LIN {X 0,Y 311.811,Z 387.645,A -85,B 0,C 180,E1 -15794.035,E2 -15794.035} C_VEL
LIN {X 0,Y 308.986,Z 387.993,A -85,B 0,C 180,E1 -15795.788,E2 -15795.788} C_VEL
LIN {X 0,Y 306.588,Z 388.29,A -85,B 0,C 180,E1 -15797.209,E2 -15797.209} C_VEL
LIN {X 0,Y 305.556,Z 388.419,A -85,B 0,C 180,E1 -15798.309,E2 -15798.309} C_VEL
LIN {X 0,Y 305.47,Z 388.429,A -85,B 0,C 180,E1 -15798.682,E2 -15798.682} C_VEL
LIN {X 0,Y 305.516,Z 388.429,A -85,B 0,C 180,E1 -15801.603,E2 -15801.603} C_VEL
LIN {X 0,Y 305.458,Z 388.434,A -85,B 0,C 180,E1 -15804.886,E2 -15804.886} C_VEL
LIN {X 0,Y 305.448,Z 388.435,A -85,B 0,C 180,E1 -15808.354,E2 -15808.354} C_VEL
LIN {X 0,Y 305.515,Z 388.427,A -85,B 0,C 180,E1 -15811.113,E2 -15811.113} C_VEL
LIN {X 0,Y 305.566,Z 388.421,A -85,B 0,C 180,E1 -15814.087,E2 -15814.087} C_VEL
LIN {X 0,Y 305.495,Z 388.428,A -85,B 0,C 180,E1 -15818.402,E2 -15818.402} C_VEL
LIN {X 0,Y 305.584,Z 388.421,A -85,B 0,C 180,E1 -15821.217,E2 -15821.217} C_VEL
LIN {X 0,Y 305.643,Z 388.415,A -85,B 0,C 180,E1 -15825.349,E2 -15825.349} C_VEL
LIN {X 0,Y 305.634,Z 388.411,A -85,B 0,C 180,E1 -15829.399,E2 -15829.399} C_VEL
LIN {X 0,Y 305.806,Z 388.39,A -85,B 0,C 180,E1 -15832.074,E2 -15832.074} C_VEL
LIN {X 0,Y 305.684,Z 388.405,A -85,B 0,C 180,E1 -15834.723,E2 -15834.723} C_VEL
LIN {X 0,Y 305.952,Z 388.373,A -85,B 0,C 180,E1 -15838.684,E2 -15838.684} C_VEL
LIN {X 0,Y 305.952,Z 388.369,A -85,B 0,C 180,E1 -15841.316,E2 -15841.316} C_VEL
LIN {X 0,Y 305.846,Z 388.386,A -85,B 0,C 180,E1 -15846.598,E2 -15846.598} C_VEL
LIN {X 0,Y 305.73,Z 388.401,A -85,B 0,C 180,E1 -15849.26,E2 -15849.26} C_VEL
LIN {X 0,Y 305.584,Z 388.416,A -85,B 0,C 180,E1 -15853.296,E2 -15853.296} C_VEL
LIN {X 0,Y 305.587,Z 388.416,A -85,B 0,C 180,E1 -15856.02,E2 -15856.02} C_VEL
LIN {X 0,Y 305.57,Z 388.416,A -85,B 0,C 180,E1 -15859.445,E2 -15859.445} C_VEL
LIN {X 0,Y 305.485,Z 388.432,A -85,B 0,C 180,E1 -15863.042,E2 -15863.042} C_VEL
LIN {X 0,Y 305.548,Z 388.422,A -85,B 0,C 180,E1 -15866.23,E2 -15866.23} C_VEL
LIN {X 0,Y 305.49,Z 388.431,A -85,B 0,C 180,E1 -15869.05,E2 -15869.05} C_VEL
LIN {X 0,Y 305.46,Z 388.429,A -85,B 0,C 180,E1 -15873.517,E2 -15873.517} C_VEL
LIN {X 0,Y 305.493,Z 388.429,A -85,B 0,C 180,E1 -15876.737,E2 -15876.737} C_VEL
LIN {X 0,Y 305.481,Z 388.431,A -85,B 0,C 180,E1 -15880.607,E2 -15880.607} C_VEL
LIN {X 0,Y 305.49,Z 388.427,A -85,B 0,C 180,E1 -15883.644,E2 -15883.644} C_VEL
LIN {X 0,Y 305.481,Z 388.431,A -85,B 0,C 180,E1 -15887.409,E2 -15887.409} C_VEL
LIN {X 0,Y 305.502,Z 388.43,A -85,B 0,C 180,E1 -15891.602,E2 -15891.602} C_VEL
LIN {X 0,Y 305.473,Z 388.437,A -85,B 0,C 180,E1 -15895.466,E2 -15895.466} C_VEL
LIN {X 0,Y 305.506,Z 388.633,A -85,B 0,C 180,E1 -15895.911,E2 -15895.911} C_VEL
LIN {X 0,Y 308.047,Z 399.573,A -85,B 0,C 180,E1 -15899.495,E2 -15899.495} C_VEL
LIN {X 0,Y 310.178,Z 410.065,A -85,B 0,C 180,E1 -15902.748,E2 -15902.748} C_VEL
LIN {X 0,Y 310.534,Z 413.788,A -85,B 0,C 180,E1 -15903.801,E2 -15903.801} C_VEL
LIN {X 0,Y 315.895,Z 444.317,A -85,B 0,C 180,E1 -15905.024,E2 -15905.024} C_VEL
LIN {X 0,Y 317.621,Z 457.948,A -85,B 0,C 180,E1 -15905.499,E2 -15905.499} C_VEL
LIN {X 0,Y 316.051,Z 522.272,A -85,B 0,C 180,E1 -15906.969,E2 -15906.969} C_VEL
LIN {X 0,Y 315.163,Z 535.447,A -85,B 0,C 180,E1 -15907.507,E2 -15907.507} C_VEL
LIN {X 0,Y 314.017,Z 547.561,A -85,B 0,C 180,E1 -15908.243,E2 -15908.243} C_VEL
LIN {X 0,Y 312.578,Z 559.793,A -85,B 0,C 180,E1 -15909.261,E2 -15909.261} C_VEL
LIN {X 0,Y 311.004,Z 571.378,A -85,B 0,C 180,E1 -15910.53,E2 -15910.53} C_VEL
LIN {X 0,Y 309.347,Z 581.811,A -85,B 0,C 180,E1 -15911.969,E2 -15911.969} C_VEL
LIN {X 0,Y 307.998,Z 591.203,A -85,B 0,C 180,E1 -15913.597,E2 -15913.597} C_VEL
LIN {X 0,Y 306.701,Z 599.615,A -85,B 0,C 180,E1 -15915.401,E2 -15915.401} C_VEL
LIN {X 0,Y 305.449,Z 607.058,A -85,B 0,C 180,E1 -15917.374,E2 -15917.374} C_VEL
LIN {X 0,Y 304.634,Z 613.044,A -85,B 0,C 180,E1 -15919.365,E2 -15919.365} C_VEL
LIN {X 0,Y 304.095,Z 617.779,A -85,B 0,C 180,E1 -15921.36,E2 -15921.36} C_VEL
LIN {X 0,Y 303.747,Z 621.398,A -85,B 0,C 180,E1 -15923.357,E2 -15923.357} C_VEL
LIN {X 0,Y 303.638,Z 623.266,A -85,B 0,C 180,E1 -15924.688,E2 -15924.688} C_VEL
LIN {X 0,Y 303.633,Z 624.67,A -85,B 0,C 180,E1 -15926.018,E2 -15926.018} C_VEL
LIN {X 0,Y 303.625,Z 625.672,A -85,B 0,C 180,E1 -15927.347,E2 -15927.347} C_VEL
LIN {X 0,Y 303.623,Z 626.282,A -85,B 0,C 180,E1 -15928.674,E2 -15928.674} C_VEL
LIN {X 0,Y 303.669,Z 626.498,A -85,B 0,C 180,E1 -15930,E2 -15930} C_VEL
LIN {X 0,Y 303.623,Z 626.275,A -85,B 0,C 180,E1 -15931.326,E2 -15931.326} C_VEL
LIN {X 0,Y 303.625,Z 625.661,A -85,B 0,C 180,E1 -15932.653,E2 -15932.653} C_VEL
LIN {X 0,Y 303.631,Z 624.656,A -85,B 0,C 180,E1 -15933.982,E2 -15933.982} C_VEL
LIN {X 0,Y 303.66,Z 622.845,A -85,B 0,C 180,E1 -15935.611,E2 -15935.611} C_VEL
LIN {X 0,Y 303.947,Z 619.055,A -85,B 0,C 180,E1 -15937.974,E2 -15937.974} C_VEL
LIN {X 0,Y 304.399,Z 614.691,A -85,B 0,C 180,E1 -15939.971,E2 -15939.971} C_VEL
LIN {X 0,Y 305.106,Z 609.138,A -85,B 0,C 180,E1 -15941.965,E2 -15941.965} C_VEL
LIN {X 0,Y 306.28,Z 602.219,A -85,B 0,C 180,E1 -15943.941,E2 -15943.941} C_VEL
LIN {X 0,Y 307.676,Z 593.562,A -85,B 0,C 180,E1 -15945.908,E2 -15945.908} C_VEL
LIN {X 0,Y 308.939,Z 584.685,A -85,B 0,C 180,E1 -15947.543,E2 -15947.543} C_VEL
LIN {X 0,Y 310.43,Z 574.952,A -85,B 0,C 180,E1 -15948.992,E2 -15948.992} C_VEL
LIN {X 0,Y 311.972,Z 564.306,A -85,B 0,C 180,E1 -15950.265,E2 -15950.265} C_VEL
LIN {X 0,Y 313.421,Z 552.402,A -85,B 0,C 180,E1 -15951.369,E2 -15951.369} C_VEL
LIN {X 0,Y 314.705,Z 540.018,A -85,B 0,C 180,E1 -15952.225,E2 -15952.225} C_VEL
LIN {X 0,Y 315.735,Z 527.279,A -85,B 0,C 180,E1 -15952.839,E2 -15952.839} C_VEL
LIN {X 0,Y 316.3,Z 513.841,A -85,B 0,C 180,E1 -15953.228,E2 -15953.228} C_VEL
LIN {X 0,Y 317.502,Z 455.967,A -85,B 0,C 180,E1 -15954.535,E2 -15954.535} C_VEL
LIN {X 0,Y 312.848,Z 426.197,A -85,B 0,C 180,E1 -15955.658,E2 -15955.658} C_VEL
LIN {X 0,Y 310.488,Z 413.594,A -85,B 0,C 180,E1 -15956.193,E2 -15956.193} C_VEL
LIN {X 0,Y 309.956,Z 408.943,A -85,B 0,C 180,E1 -15957.568,E2 -15957.568} C_VEL
LIN {X 0,Y 308.048,Z 399.473,A -85,B 0,C 180,E1 -15960.505,E2 -15960.505} C_VEL
LIN {X 0,Y 305.466,Z 388.438,A -85,B 0,C 180,E1 -15964.131,E2 -15964.131} C_VEL
LIN {X 0,Y 305.495,Z 388.432,A -85,B 0,C 180,E1 -15966.736,E2 -15966.736} C_VEL
LIN {X 0,Y 305.455,Z 388.434,A -85,B 0,C 180,E1 -15970.6,E2 -15970.6} C_VEL
LIN {X 0,Y 305.468,Z 388.432,A -85,B 0,C 180,E1 -15973.646,E2 -15973.646} C_VEL
LIN {X 0,Y 305.505,Z 388.429,A -85,B 0,C 180,E1 -15977.403,E2 -15977.403} C_VEL
LIN {X 0,Y 305.506,Z 388.43,A -85,B 0,C 180,E1 -15981.602,E2 -15981.602} C_VEL
LIN {X 0,Y 305.458,Z 388.435,A -85,B 0,C 180,E1 -15984.886,E2 -15984.886} C_VEL
LIN {X 0,Y 305.447,Z 388.434,A -85,B 0,C 180,E1 -15988.354,E2 -15988.354} C_VEL
LIN {X 0,Y 305.516,Z 388.426,A -85,B 0,C 180,E1 -15991.113,E2 -15991.113} C_VEL
LIN {X 0,Y 305.567,Z 388.419,A -85,B 0,C 180,E1 -15994.087,E2 -15994.087} C_VEL
LIN {X 0,Y 305.494,Z 388.427,A -85,B 0,C 180,E1 -15998.402,E2 -15998.402} C_VEL
LIN {X 0,Y 305.584,Z 388.419,A -85,B 0,C 180,E1 -16001.217,E2 -16001.217} C_VEL
LIN {X 0,Y 305.643,Z 388.414,A -85,B 0,C 180,E1 -16005.349,E2 -16005.349} C_VEL
LIN {X 0,Y 305.634,Z 388.408,A -85,B 0,C 180,E1 -16009.4,E2 -16009.4} C_VEL
LIN {X 0,Y 305.806,Z 388.389,A -85,B 0,C 180,E1 -16012.074,E2 -16012.074} C_VEL
LIN {X 0,Y 305.684,Z 388.408,A -85,B 0,C 180,E1 -16014.723,E2 -16014.723} C_VEL
LIN {X 0,Y 305.952,Z 388.37,A -85,B 0,C 180,E1 -16018.684,E2 -16018.684} C_VEL
LIN {X 0,Y 305.952,Z 388.373,A -85,B 0,C 180,E1 -16021.316,E2 -16021.316} C_VEL
LIN {X 0,Y 305.846,Z 388.384,A -85,B 0,C 180,E1 -16026.598,E2 -16026.598} C_VEL
LIN {X 0,Y 305.73,Z 388.4,A -85,B 0,C 180,E1 -16029.26,E2 -16029.26} C_VEL
LIN {X 0,Y 305.584,Z 388.416,A -85,B 0,C 180,E1 -16033.296,E2 -16033.296} C_VEL
LIN {X 0,Y 305.588,Z 388.418,A -85,B 0,C 180,E1 -16036.021,E2 -16036.021} C_VEL
LIN {X 0,Y 305.571,Z 388.414,A -85,B 0,C 180,E1 -16039.445,E2 -16039.445} C_VEL
LIN {X 0,Y 305.485,Z 388.432,A -85,B 0,C 180,E1 -16043.042,E2 -16043.042} C_VEL
LIN {X 0,Y 305.542,Z 388.42,A -85,B 0,C 180,E1 -16046.228,E2 -16046.228} C_VEL
LIN {X 0,Y 305.491,Z 388.431,A -85,B 0,C 180,E1 -16049.05,E2 -16049.05} C_VEL
LIN {X 0,Y 305.46,Z 388.433,A -85,B 0,C 180,E1 -16053.518,E2 -16053.518} C_VEL
LIN {X 0,Y 305.498,Z 388.429,A -85,B 0,C 180,E1 -16056.736,E2 -16056.736} C_VEL
LIN {X 0,Y 305.482,Z 388.431,A -85,B 0,C 180,E1 -16060.607,E2 -16060.607} C_VEL
LIN {X 0,Y 305.49,Z 388.43,A -85,B 0,C 180,E1 -16063.644,E2 -16063.644} C_VEL
LIN {X 0,Y 305.461,Z 388.433,A -85,B 0,C 180,E1 -16067.413,E2 -16067.413} C_VEL
LIN {X 0,Y 305.494,Z 388.43,A -85,B 0,C 180,E1 -16071.601,E2 -16071.601} C_VEL
LIN {X 0,Y 305.462,Z 388.435,A -85,B 0,C 180,E1 -16074.888,E2 -16074.888} C_VEL
LIN {X 0,Y 305.45,Z 388.439,A -85,B 0,C 180,E1 -16078.356,E2 -16078.356} C_VEL
LIN {X 0,Y 305.542,Z 388.49,A -85,B 0,C 180,E1 -16081.68,E2 -16081.68} C_VEL
LIN {X 0,Y 306.681,Z 393.494,A -85,B 0,C 180,E1 -16083.529,E2 -16083.529} C_VEL
LIN {X 0,Y 315.952,Z 416.268,A -85,B 0,C 180,E1 -16084.939,E2 -16084.939} C_VEL
LIN {X 0,Y 317.657,Z 421.102,A -85,B 0,C 180,E1 -16085.203,E2 -16085.203} C_VEL
LIN {X 0,Y 318.311,Z 425.219,A -85,B 0,C 180,E1 -16085.358,E2 -16085.358} C_VEL
LIN {X 0,Y 316.452,Z 500.83,A -85,B 0,C 180,E1 -16087.087,E2 -16087.087} C_VEL
LIN {X 0,Y 315.602,Z 514.574,A -85,B 0,C 180,E1 -16087.67,E2 -16087.67} C_VEL
LIN {X 0,Y 314.661,Z 526.897,A -85,B 0,C 180,E1 -16088.462,E2 -16088.462} C_VEL
LIN {X 0,Y 313.426,Z 538.705,A -85,B 0,C 180,E1 -16089.491,E2 -16089.491} C_VEL
LIN {X 0,Y 311.975,Z 550.046,A -85,B 0,C 180,E1 -16090.765,E2 -16090.765} C_VEL
LIN {X 0,Y 310.648,Z 560.751,A -85,B 0,C 180,E1 -16092.303,E2 -16092.303} C_VEL
LIN {X 0,Y 309.2,Z 569.411,A -85,B 0,C 180,E1 -16093.833,E2 -16093.833} C_VEL
LIN {X 0,Y 307.641,Z 578.311,A -85,B 0,C 180,E1 -16095.784,E2 -16095.784} C_VEL
LIN {X 0,Y 306.435,Z 585.47,A -85,B 0,C 180,E1 -16097.752,E2 -16097.752} C_VEL
LIN {X 0,Y 305.596,Z 590.296,A -85,B 0,C 180,E1 -16099.398,E2 -16099.398} C_VEL
LIN {X 0,Y 304.832,Z 594.983,A -85,B 0,C 180,E1 -16101.381,E2 -16101.381} C_VEL
LIN {X 0,Y 304.35,Z 598.567,A -85,B 0,C 180,E1 -16103.37,E2 -16103.37} C_VEL
LIN {X 0,Y 304.119,Z 600.418,A -85,B 0,C 180,E1 -16104.696,E2 -16104.696} C_VEL
LIN {X 0,Y 303.925,Z 601.811,A -85,B 0,C 180,E1 -16106.022,E2 -16106.022} C_VEL
LIN {X 0,Y 303.682,Z 603.413,A -85,B 0,C 180,E1 -16108.674,E2 -16108.674} C_VEL
LIN {X 0,Y 303.677,Z 603.643,A -85,B 0,C 180,E1 -16110,E2 -16110} C_VEL
LIN {X 0,Y 303.682,Z 603.452,A -85,B 0,C 180,E1 -16111.326,E2 -16111.326} C_VEL
LIN {X 0,Y 303.924,Z 601.901,A -85,B 0,C 180,E1 -16113.978,E2 -16113.978} C_VEL
LIN {X 0,Y 304.118,Z 600.547,A -85,B 0,C 180,E1 -16115.304,E2 -16115.304} C_VEL
LIN {X 0,Y 304.472,Z 598.158,A -85,B 0,C 180,E1 -16116.995,E2 -16116.995} C_VEL
LIN {X 0,Y 305.019,Z 593.81,A -85,B 0,C 180,E1 -16119.281,E2 -16119.281} C_VEL
LIN {X 0,Y 305.887,Z 588.801,A -85,B 0,C 180,E1 -16121.262,E2 -16121.262} C_VEL
LIN {X 0,Y 306.971,Z 582.493,A -85,B 0,C 180,E1 -16123.235,E2 -16123.235} C_VEL
LIN {X 0,Y 308.267,Z 574.597,A -85,B 0,C 180,E1 -16125.199,E2 -16125.199} C_VEL
LIN {X 0,Y 309.691,Z 566.539,A -85,B 0,C 180,E1 -16126.818,E2 -16126.818} C_VEL
LIN {X 0,Y 311.094,Z 556.711,A -85,B 0,C 180,E1 -16128.438,E2 -16128.438} C_VEL
LIN {X 0,Y 312.554,Z 545.645,A -85,B 0,C 180,E1 -16129.882,E2 -16129.882} C_VEL
LIN {X 0,Y 314.119,Z 533.028,A -85,B 0,C 180,E1 -16131.147,E2 -16131.147} C_VEL
LIN {X 0,Y 315.312,Z 520.402,A -85,B 0,C 180,E1 -16132.093,E2 -16132.093} C_VEL
LIN {X 0,Y 316.15,Z 507.737,A -85,B 0,C 180,E1 -16132.764,E2 -16132.764} C_VEL
LIN {X 0,Y 316.692,Z 494.689,A -85,B 0,C 180,E1 -16133.197,E2 -16133.197} C_VEL
LIN {X 0,Y 318.267,Z 423.968,A -85,B 0,C 180,E1 -16134.79,E2 -16134.79} C_VEL
LIN {X 0,Y 316.849,Z 418.647,A -85,B 0,C 180,E1 -16135.041,E2 -16135.041} C_VEL
LIN {X 0,Y 309.15,Z 399.307,A -85,B 0,C 180,E1 -16136.207,E2 -16136.207} C_VEL
LIN {X 0,Y 306.686,Z 393.484,A -85,B 0,C 180,E1 -16136.596,E2 -16136.596} C_VEL
LIN {X 0,Y 305.522,Z 388.43,A -85,B 0,C 180,E1 -16138.51,E2 -16138.51} C_VEL
LIN {X 0,Y 305.443,Z 388.441,A -85,B 0,C 180,E1 -16141.951,E2 -16141.951} C_VEL
LIN {X 0,Y 305.462,Z 388.435,A -85,B 0,C 180,E1 -16145.112,E2 -16145.112} C_VEL
LIN {X 0,Y 305.465,Z 388.434,A -85,B 0,C 180,E1 -16148.532,E2 -16148.532} C_VEL
LIN {X 0,Y 305.461,Z 388.432,A -85,B 0,C 180,E1 -16152.587,E2 -16152.587} C_VEL
LIN {X 0,Y 305.49,Z 388.424,A -85,B 0,C 180,E1 -16156.356,E2 -16156.356} C_VEL
LIN {X 0,Y 305.47,Z 388.429,A -85,B 0,C 180,E1 -16158.682,E2 -16158.682} C_VEL
LIN {X 0,Y 304.799,Z 388.519,A -85,B 0,C 180,E1 -16159.783,E2 -16159.783} C_VEL
LIN {X 0,Y 301.949,Z 388.874,A -85,B 0,C 180,E1 -16161.576,E2 -16161.576} C_VEL
LIN {X 0,Y 299.532,Z 389.174,A -85,B 0,C 180,E1 -16163.03,E2 -16163.03} C_VEL
LIN {X 0,Y 298.489,Z 389.303,A -85,B 0,C 180,E1 -16164.156,E2 -16164.156} C_VEL
LIN {X 0,Y 298.401,Z 389.312,A -85,B 0,C 180,E1 -16164.537,E2 -16164.537} C_VEL
LIN {X 0,Y 298.391,Z 389.314,A -85,B 0,C 180,E1 -16168.791,E2 -16168.791} C_VEL
LIN {X 0,Y 298.458,Z 389.306,A -85,B 0,C 180,E1 -16171.904,E2 -16171.904} C_VEL
LIN {X 0,Y 298.48,Z 389.304,A -85,B 0,C 180,E1 -16174.923,E2 -16174.923} C_VEL
LIN {X 0,Y 298.445,Z 389.311,A -85,B 0,C 180,E1 -16179.315,E2 -16179.315} C_VEL
LIN {X 0,Y 298.532,Z 389.292,A -85,B 0,C 180,E1 -16182.179,E2 -16182.179} C_VEL
LIN {X 0,Y 298.587,Z 389.291,A -85,B 0,C 180,E1 -16184.994,E2 -16184.994} C_VEL
LIN {X 0,Y 298.589,Z 389.287,A -85,B 0,C 180,E1 -16189.146,E2 -16189.146} C_VEL
LIN {X 0,Y 298.752,Z 389.269,A -85,B 0,C 180,E1 -16191.886,E2 -16191.886} C_VEL
LIN {X 0,Y 298.655,Z 389.279,A -85,B 0,C 180,E1 -16194.599,E2 -16194.599} C_VEL
LIN {X 0,Y 298.919,Z 389.249,A -85,B 0,C 180,E1 -16198.653,E2 -16198.653} C_VEL
LIN {X 0,Y 298.919,Z 389.244,A -85,B 0,C 180,E1 -16201.347,E2 -16201.347} C_VEL
LIN {X 0,Y 298.791,Z 389.266,A -85,B 0,C 180,E1 -16206.754,E2 -16206.754} C_VEL
LIN {X 0,Y 298.675,Z 389.278,A -85,B 0,C 180,E1 -16209.481,E2 -16209.481} C_VEL
LIN {X 0,Y 298.547,Z 389.29,A -85,B 0,C 180,E1 -16213.616,E2 -16213.616} C_VEL
LIN {X 0,Y 298.542,Z 389.295,A -85,B 0,C 180,E1 -16216.409,E2 -16216.409} C_VEL
LIN {X 0,Y 298.505,Z 389.295,A -85,B 0,C 180,E1 -16219.655,E2 -16219.655} C_VEL
LIN {X 0,Y 298.452,Z 389.305,A -85,B 0,C 180,E1 -16223.598,E2 -16223.598} C_VEL
LIN {X 0,Y 298.487,Z 389.305,A -85,B 0,C 180,E1 -16226.575,E2 -16226.575} C_VEL
LIN {X 0,Y 298.416,Z 389.31,A -85,B 0,C 180,E1 -16229.642,E2 -16229.642} C_VEL
LIN {X 0,Y 298.391,Z 389.313,A -85,B 0,C 180,E1 -16232.801,E2 -16232.801} C_VEL
LIN {X 0,Y 298.462,Z 389.304,A -85,B 0,C 180,E1 -16236.813,E2 -16236.813} C_VEL
LIN {X 0,Y 298.448,Z 389.306,A -85,B 0,C 180,E1 -16241.251,E2 -16241.251} C_VEL
LIN {X 0,Y 298.414,Z 389.312,A -85,B 0,C 180,E1 -16245.048,E2 -16245.048} C_VEL
LIN {X 0,Y 298.411,Z 389.314,A -85,B 0,C 180,E1 -16248.907,E2 -16248.907} C_VEL
LIN {X 0,Y 298.463,Z 389.309,A -85,B 0,C 180,E1 -16253.188,E2 -16253.188} C_VEL
LIN {X 0,Y 298.446,Z 389.483,A -85,B 0,C 180,E1 -16255.347,E2 -16255.347} C_VEL
LIN {X 0,Y 301.028,Z 400.576,A -85,B 0,C 180,E1 -16259.095,E2 -16259.095} C_VEL
LIN {X 0,Y 303.14,Z 410.847,A -85,B 0,C 180,E1 -16262.376,E2 -16262.376} C_VEL
LIN {X 0,Y 303.577,Z 413.519,A -85,B 0,C 180,E1 -16263.153,E2 -16263.153} C_VEL
LIN {X 0,Y 305.073,Z 419.768,A -85,B 0,C 180,E1 -16263.455,E2 -16263.455} C_VEL
LIN {X 0,Y 309.974,Z 448.85,A -85,B 0,C 180,E1 -16264.633,E2 -16264.633} C_VEL
LIN {X 0,Y 311.143,Z 458.683,A -85,B 0,C 180,E1 -16264.979,E2 -16264.979} C_VEL
LIN {X 0,Y 309.541,Z 522.018,A -85,B 0,C 180,E1 -16266.456,E2 -16266.456} C_VEL
LIN {X 0,Y 308.55,Z 535.952,A -85,B 0,C 180,E1 -16267.042,E2 -16267.042} C_VEL
LIN {X 0,Y 307.29,Z 548.414,A -85,B 0,C 180,E1 -16267.83,E2 -16267.83} C_VEL
LIN {X 0,Y 305.933,Z 559.53,A -85,B 0,C 180,E1 -16268.789,E2 -16268.789} C_VEL
LIN {X 0,Y 304.305,Z 571.114,A -85,B 0,C 180,E1 -16270.084,E2 -16270.084} C_VEL
LIN {X 0,Y 302.586,Z 581.546,A -85,B 0,C 180,E1 -16271.551,E2 -16271.551} C_VEL
LIN {X 0,Y 301.2,Z 590.232,A -85,B 0,C 180,E1 -16273.072,E2 -16273.072} C_VEL
LIN {X 0,Y 300.003,Z 597.968,A -85,B 0,C 180,E1 -16274.72,E2 -16274.72} C_VEL
LIN {X 0,Y 298.722,Z 605.669,A -85,B 0,C 180,E1 -16276.739,E2 -16276.739} C_VEL
LIN {X 0,Y 297.855,Z 610.949,A -85,B 0,C 180,E1 -16278.431,E2 -16278.431} C_VEL
LIN {X 0,Y 297.204,Z 616.073,A -85,B 0,C 180,E1 -16280.472,E2 -16280.472} C_VEL
LIN {X 0,Y 296.786,Z 620.055,A -85,B 0,C 180,E1 -16282.517,E2 -16282.517} C_VEL
LIN {X 0,Y 296.552,Z 622.999,A -85,B 0,C 180,E1 -16284.561,E2 -16284.561} C_VEL
LIN {X 0,Y 296.531,Z 624.403,A -85,B 0,C 180,E1 -16285.923,E2 -16285.923} C_VEL
LIN {X 0,Y 296.55,Z 625.405,A -85,B 0,C 180,E1 -16287.283,E2 -16287.283} C_VEL
LIN {X 0,Y 296.54,Z 626.016,A -85,B 0,C 180,E1 -16288.642,E2 -16288.642} C_VEL
LIN {X 0,Y 296.581,Z 626.232,A -85,B 0,C 180,E1 -16290,E2 -16290} C_VEL
LIN {X 0,Y 296.54,Z 626.008,A -85,B 0,C 180,E1 -16291.358,E2 -16291.358} C_VEL
LIN {X 0,Y 296.55,Z 625.394,A -85,B 0,C 180,E1 -16292.717,E2 -16292.717} C_VEL
LIN {X 0,Y 296.529,Z 624.388,A -85,B 0,C 180,E1 -16294.077,E2 -16294.077} C_VEL
LIN {X 0,Y 296.553,Z 622.872,A -85,B 0,C 180,E1 -16295.523,E2 -16295.523} C_VEL
LIN {X 0,Y 296.888,Z 618.785,A -85,B 0,C 180,E1 -16298.165,E2 -16298.165} C_VEL
LIN {X 0,Y 297.385,Z 614.422,A -85,B 0,C 180,E1 -16300.209,E2 -16300.209} C_VEL
LIN {X 0,Y 298.129,Z 608.868,A -85,B 0,C 180,E1 -16302.249,E2 -16302.249} C_VEL
LIN {X 0,Y 299.376,Z 601.95,A -85,B 0,C 180,E1 -16304.27,E2 -16304.27} C_VEL
LIN {X 0,Y 300.554,Z 594.885,A -85,B 0,C 180,E1 -16305.947,E2 -16305.947} C_VEL
LIN {X 0,Y 301.856,Z 586.37,A -85,B 0,C 180,E1 -16307.618,E2 -16307.618} C_VEL
LIN {X 0,Y 303.328,Z 577.035,A -85,B 0,C 180,E1 -16309.103,E2 -16309.103} C_VEL
LIN {X 0,Y 305.08,Z 565.464,A -85,B 0,C 180,E1 -16310.567,E2 -16310.567} C_VEL
LIN {X 0,Y 306.631,Z 554.068,A -85,B 0,C 180,E1 -16311.69,E2 -16311.69} C_VEL
LIN {X 0,Y 307.927,Z 542.349,A -85,B 0,C 180,E1 -16312.564,E2 -16312.564} C_VEL
LIN {X 0,Y 309.024,Z 529.756,A -85,B 0,C 180,E1 -16313.231,E2 -16313.231} C_VEL
LIN {X 0,Y 309.691,Z 516.923,A -85,B 0,C 180,E1 -16313.665,E2 -16313.665} C_VEL
LIN {X 0,Y 311.047,Z 457.003,A -85,B 0,C 180,E1 -16315.046,E2 -16315.046} C_VEL
LIN {X 0,Y 306.608,Z 428.099,A -85,B 0,C 180,E1 -16316.164,E2 -16316.164} C_VEL
LIN {X 0,Y 303.846,Z 414.488,A -85,B 0,C 180,E1 -16316.768,E2 -16316.768} C_VEL
LIN {X 0,Y 303.518,Z 413.158,A -85,B 0,C 180,E1 -16316.886,E2 -16316.886} C_VEL
LIN {X 0,Y 301.807,Z 403.876,A -85,B 0,C 180,E1 -16319.798,E2 -16319.798} C_VEL
LIN {X 0,Y 299.204,Z 392.71,A -85,B 0,C 180,E1 -16323.503,E2 -16323.503} C_VEL
LIN {X 0,Y 298.424,Z 389.315,A -85,B 0,C 180,E1 -16324.712,E2 -16324.712} C_VEL
LIN {X 0,Y 298.435,Z 389.308,A -85,B 0,C 180,E1 -16327.754,E2 -16327.754} C_VEL
LIN {X 0,Y 298.412,Z 389.314,A -85,B 0,C 180,E1 -16331.256,E2 -16331.256} C_VEL
LIN {X 0,Y 298.414,Z 389.304,A -85,B 0,C 180,E1 -16335.046,E2 -16335.046} C_VEL
LIN {X 0,Y 298.448,Z 389.306,A -85,B 0,C 180,E1 -16338.749,E2 -16338.749} C_VEL
LIN {X 0,Y 298.462,Z 389.306,A -85,B 0,C 180,E1 -16343.187,E2 -16343.187} C_VEL
LIN {X 0,Y 298.391,Z 389.313,A -85,B 0,C 180,E1 -16347.199,E2 -16347.199} C_VEL
LIN {X 0,Y 298.464,Z 389.302,A -85,B 0,C 180,E1 -16351.904,E2 -16351.904} C_VEL
LIN {X 0,Y 298.48,Z 389.304,A -85,B 0,C 180,E1 -16354.924,E2 -16354.924} C_VEL
LIN {X 0,Y 298.444,Z 389.311,A -85,B 0,C 180,E1 -16359.315,E2 -16359.315} C_VEL
LIN {X 0,Y 298.531,Z 389.292,A -85,B 0,C 180,E1 -16362.179,E2 -16362.179} C_VEL
LIN {X 0,Y 298.587,Z 389.29,A -85,B 0,C 180,E1 -16364.994,E2 -16364.994} C_VEL
LIN {X 0,Y 298.589,Z 389.286,A -85,B 0,C 180,E1 -16369.146,E2 -16369.146} C_VEL
LIN {X 0,Y 298.751,Z 389.268,A -85,B 0,C 180,E1 -16371.886,E2 -16371.886} C_VEL
LIN {X 0,Y 298.655,Z 389.283,A -85,B 0,C 180,E1 -16374.599,E2 -16374.599} C_VEL
LIN {X 0,Y 298.919,Z 389.245,A -85,B 0,C 180,E1 -16378.653,E2 -16378.653} C_VEL
LIN {X 0,Y 298.919,Z 389.249,A -85,B 0,C 180,E1 -16381.347,E2 -16381.347} C_VEL
LIN {X 0,Y 298.791,Z 389.264,A -85,B 0,C 180,E1 -16386.754,E2 -16386.754} C_VEL
LIN {X 0,Y 298.675,Z 389.278,A -85,B 0,C 180,E1 -16389.481,E2 -16389.481} C_VEL
LIN {X 0,Y 298.547,Z 389.291,A -85,B 0,C 180,E1 -16393.616,E2 -16393.616} C_VEL
LIN {X 0,Y 298.543,Z 389.298,A -85,B 0,C 180,E1 -16396.409,E2 -16396.409} C_VEL
LIN {X 0,Y 298.506,Z 389.293,A -85,B 0,C 180,E1 -16399.655,E2 -16399.655} C_VEL
LIN {X 0,Y 298.452,Z 389.306,A -85,B 0,C 180,E1 -16403.598,E2 -16403.598} C_VEL
LIN {X 0,Y 298.485,Z 389.301,A -85,B 0,C 180,E1 -16406.575,E2 -16406.575} C_VEL
LIN {X 0,Y 298.416,Z 389.311,A -85,B 0,C 180,E1 -16409.642,E2 -16409.642} C_VEL
LIN {X 0,Y 298.391,Z 389.316,A -85,B 0,C 180,E1 -16412.801,E2 -16412.801} C_VEL
LIN {X 0,Y 298.466,Z 389.304,A -85,B 0,C 180,E1 -16416.814,E2 -16416.814} C_VEL
LIN {X 0,Y 298.449,Z 389.304,A -85,B 0,C 180,E1 -16421.251,E2 -16421.251} C_VEL
LIN {X 0,Y 298.414,Z 389.31,A -85,B 0,C 180,E1 -16425.048,E2 -16425.048} C_VEL
LIN {X 0,Y 298.386,Z 389.316,A -85,B 0,C 180,E1 -16428.913,E2 -16428.913} C_VEL
LIN {X 0,Y 298.464,Z 389.306,A -85,B 0,C 180,E1 -16433.188,E2 -16433.188} C_VEL
LIN {X 0,Y 298.395,Z 389.315,A -85,B 0,C 180,E1 -16437.201,E2 -16437.201} C_VEL
LIN {X 0,Y 298.47,Z 389.31,A -85,B 0,C 180,E1 -16441.138,E2 -16441.138} C_VEL
LIN {X 0,Y 299.603,Z 394.019,A -85,B 0,C 180,E1 -16442.861,E2 -16442.861} C_VEL
LIN {X 0,Y 308.112,Z 414.287,A -85,B 0,C 180,E1 -16444.196,E2 -16444.196} C_VEL
LIN {X 0,Y 311.401,Z 423.085,A -85,B 0,C 180,E1 -16444.712,E2 -16444.712} C_VEL
LIN {X 0,Y 311.875,Z 425.907,A -85,B 0,C 180,E1 -16444.825,E2 -16444.825} C_VEL
LIN {X 0,Y 309.946,Z 501.112,A -85,B 0,C 180,E1 -16446.577,E2 -16446.577} C_VEL
LIN {X 0,Y 309.06,Z 514.851,A -85,B 0,C 180,E1 -16447.17,E2 -16447.17} C_VEL
LIN {X 0,Y 308.092,Z 527.17,A -85,B 0,C 180,E1 -16447.979,E2 -16447.979} C_VEL
LIN {X 0,Y 306.788,Z 538.978,A -85,B 0,C 180,E1 -16449.027,E2 -16449.027} C_VEL
LIN {X 0,Y 305.274,Z 550.318,A -85,B 0,C 180,E1 -16450.325,E2 -16450.325} C_VEL
LIN {X 0,Y 304.06,Z 559.834,A -85,B 0,C 180,E1 -16451.705,E2 -16451.705} C_VEL
LIN {X 0,Y 302.649,Z 567.993,A -85,B 0,C 180,E1 -16453.126,E2 -16453.126} C_VEL
LIN {X 0,Y 301.296,Z 575.848,A -85,B 0,C 180,E1 -16454.787,E2 -16454.787} C_VEL
LIN {X 0,Y 299.886,Z 583.523,A -85,B 0,C 180,E1 -16456.792,E2 -16456.792} C_VEL
LIN {X 0,Y 298.63,Z 590.564,A -85,B 0,C 180,E1 -16459.148,E2 -16459.148} C_VEL
LIN {X 0,Y 297.803,Z 595.252,A -85,B 0,C 180,E1 -16461.176,E2 -16461.176} C_VEL
LIN {X 0,Y 297.301,Z 598.835,A -85,B 0,C 180,E1 -16463.212,E2 -16463.212} C_VEL
LIN {X 0,Y 297.057,Z 600.686,A -85,B 0,C 180,E1 -16464.57,E2 -16464.57} C_VEL
LIN {X 0,Y 296.865,Z 602.078,A -85,B 0,C 180,E1 -16465.927,E2 -16465.927} C_VEL
LIN {X 0,Y 296.598,Z 603.68,A -85,B 0,C 180,E1 -16468.642,E2 -16468.642} C_VEL
LIN {X 0,Y 296.589,Z 603.909,A -85,B 0,C 180,E1 -16470,E2 -16470} C_VEL
LIN {X 0,Y 296.598,Z 603.719,A -85,B 0,C 180,E1 -16471.358,E2 -16471.358} C_VEL
LIN {X 0,Y 296.864,Z 602.167,A -85,B 0,C 180,E1 -16474.073,E2 -16474.073} C_VEL
LIN {X 0,Y 297.057,Z 600.814,A -85,B 0,C 180,E1 -16475.43,E2 -16475.43} C_VEL
LIN {X 0,Y 297.489,Z 597.954,A -85,B 0,C 180,E1 -16477.465,E2 -16477.465} C_VEL
LIN {X 0,Y 298.03,Z 594.076,A -85,B 0,C 180,E1 -16479.501,E2 -16479.501} C_VEL
LIN {X 0,Y 298.94,Z 589.066,A -85,B 0,C 180,E1 -16481.527,E2 -16481.527} C_VEL
LIN {X 0,Y 300.07,Z 582.758,A -85,B 0,C 180,E1 -16483.545,E2 -16483.545} C_VEL
LIN {X 0,Y 301.434,Z 574.861,A -85,B 0,C 180,E1 -16485.552,E2 -16485.552} C_VEL
LIN {X 0,Y 302.903,Z 566.803,A -85,B 0,C 180,E1 -16487.207,E2 -16487.207} C_VEL
LIN {X 0,Y 304.378,Z 556.974,A -85,B 0,C 180,E1 -16488.859,E2 -16488.859} C_VEL
LIN {X 0,Y 305.908,Z 545.907,A -85,B 0,C 180,E1 -16490.333,E2 -16490.333} C_VEL
LIN {X 0,Y 307.524,Z 533.288,A -85,B 0,C 180,E1 -16491.623,E2 -16491.623} C_VEL
LIN {X 0,Y 308.761,Z 520.659,A -85,B 0,C 180,E1 -16492.588,E2 -16492.588} C_VEL
LIN {X 0,Y 309.634,Z 507.991,A -85,B 0,C 180,E1 -16493.271,E2 -16493.271} C_VEL
LIN {X 0,Y 310.199,Z 494.935,A -85,B 0,C 180,E1 -16493.712,E2 -16493.712} C_VEL
LIN {X 0,Y 311.846,Z 425.247,A -85,B 0,C 180,E1 -16495.31,E2 -16495.31} C_VEL
LIN {X 0,Y 310.389,Z 420.239,A -85,B 0,C 180,E1 -16495.565,E2 -16495.565} C_VEL
LIN {X 0,Y 303.195,Z 402.289,A -85,B 0,C 180,E1 -16496.69,E2 -16496.69} C_VEL
LIN {X 0,Y 299.519,Z 393.747,A -85,B 0,C 180,E1 -16497.296,E2 -16497.296} C_VEL
LIN {X 0,Y 298.47,Z 389.308,A -85,B 0,C 180,E1 -16498.991,E2 -16498.991} C_VEL
LIN {X 0,Y 298.395,Z 389.316,A -85,B 0,C 180,E1 -16502.799,E2 -16502.799} C_VEL
LIN {X 0,Y 298.463,Z 389.306,A -85,B 0,C 180,E1 -16506.811,E2 -16506.811} C_VEL
LIN {X 0,Y 298.386,Z 389.315,A -85,B 0,C 180,E1 -16511.087,E2 -16511.087} C_VEL
LIN {X 0,Y 298.414,Z 389.311,A -85,B 0,C 180,E1 -16514.952,E2 -16514.952} C_VEL
LIN {X 0,Y 298.449,Z 389.303,A -85,B 0,C 180,E1 -16518.749,E2 -16518.749} C_VEL
LIN {X 0,Y 298.466,Z 389.303,A -85,B 0,C 180,E1 -16523.186,E2 -16523.186} C_VEL
LIN {X 0,Y 298.401,Z 389.312,A -85,B 0,C 180,E1 -16524.537,E2 -16524.537} C_VEL
LIN {X 0,Y 297.73,Z 389.398,A -85,B 0,C 180,E1 -16525.663,E2 -16525.663} C_VEL
LIN {X 0,Y 294.899,Z 389.749,A -85,B 0,C 180,E1 -16527.498,E2 -16527.498} C_VEL
LIN {X 0,Y 292.498,Z 390.049,A -85,B 0,C 180,E1 -16528.986,E2 -16528.986} C_VEL
LIN {X 0,Y 291.462,Z 390.177,A -85,B 0,C 180,E1 -16530.138,E2 -16530.138} C_VEL
LIN {X 0,Y 291.374,Z 390.186,A -85,B 0,C 180,E1 -16530.528,E2 -16530.528} C_VEL
LIN {X 0,Y 291.411,Z 390.184,A -85,B 0,C 180,E1 -16534.271,E2 -16534.271} C_VEL
LIN {X 0,Y 291.376,Z 390.186,A -85,B 0,C 180,E1 -16537.299,E2 -16537.299} C_VEL
LIN {X 0,Y 291.453,Z 390.178,A -85,B 0,C 180,E1 -16540.27,E2 -16540.27} C_VEL
LIN {X 0,Y 291.535,Z 390.167,A -85,B 0,C 180,E1 -16544.634,E2 -16544.634} C_VEL
LIN {X 0,Y 291.532,Z 390.165,A -85,B 0,C 180,E1 -16548.88,E2 -16548.88} C_VEL
LIN {X 0,Y 291.703,Z 390.149,A -85,B 0,C 180,E1 -16551.688,E2 -16551.688} C_VEL
LIN {X 0,Y 291.625,Z 390.154,A -85,B 0,C 180,E1 -16554.468,E2 -16554.468} C_VEL
LIN {X 0,Y 291.885,Z 390.125,A -85,B 0,C 180,E1 -16558.62,E2 -16558.62} C_VEL
LIN {X 0,Y 291.885,Z 390.12,A -85,B 0,C 180,E1 -16561.38,E2 -16561.38} C_VEL
LIN {X 0,Y 291.74,Z 390.143,A -85,B 0,C 180,E1 -16566.918,E2 -16566.918} C_VEL
LIN {X 0,Y 291.624,Z 390.155,A -85,B 0,C 180,E1 -16569.712,E2 -16569.712} C_VEL
LIN {X 0,Y 291.517,Z 390.165,A -85,B 0,C 180,E1 -16573.951,E2 -16573.951} C_VEL
LIN {X 0,Y 291.481,Z 390.178,A -85,B 0,C 180,E1 -16576.818,E2 -16576.818} C_VEL
LIN {X 0,Y 291.445,Z 390.174,A -85,B 0,C 180,E1 -16579.875,E2 -16579.875} C_VEL
LIN {X 0,Y 291.395,Z 390.185,A -85,B 0,C 180,E1 -16584.206,E2 -16584.206} C_VEL
LIN {X 0,Y 291.421,Z 390.183,A -85,B 0,C 180,E1 -16587.272,E2 -16587.272} C_VEL
LIN {X 0,Y 291.332,Z 390.195,A -85,B 0,C 180,E1 -16590.437,E2 -16590.437} C_VEL
LIN {X 0,Y 291.34,Z 390.188,A -85,B 0,C 180,E1 -16593.699,E2 -16593.699} C_VEL
LIN {X 0,Y 291.395,Z 390.182,A -85,B 0,C 180,E1 -16597.261,E2 -16597.261} C_VEL
LIN {X 0,Y 291.397,Z 390.185,A -85,B 0,C 180,E1 -16600.632,E2 -16600.632} C_VEL
LIN {X 0,Y 291.35,Z 390.192,A -85,B 0,C 180,E1 -16604.39,E2 -16604.39} C_VEL
LIN {X 0,Y 291.35,Z 390.193,A -85,B 0,C 180,E1 -16608.399,E2 -16608.399} C_VEL
LIN {X 0,Y 291.369,Z 390.191,A -85,B 0,C 180,E1 -16611.162,E2 -16611.162} C_VEL
LIN {X 0,Y 291.413,Z 390.28,A -85,B 0,C 180,E1 -16614.742,E2 -16614.742} C_VEL
LIN {X 0,Y 294.139,Z 402.161,A -85,B 0,C 180,E1 -16618.875,E2 -16618.875} C_VEL
LIN {X 0,Y 296.366,Z 413.077,A -85,B 0,C 180,E1 -16622.441,E2 -16622.441} C_VEL
LIN {X 0,Y 298.52,Z 419.743,A -85,B 0,C 180,E1 -16622.831,E2 -16622.831} C_VEL
LIN {X 0,Y 303.615,Z 450.19,A -85,B 0,C 180,E1 -16624.103,E2 -16624.103} C_VEL
LIN {X 0,Y 304.691,Z 459.382,A -85,B 0,C 180,E1 -16624.435,E2 -16624.435} C_VEL
LIN {X 0,Y 303.051,Z 521.765,A -85,B 0,C 180,E1 -16625.921,E2 -16625.921} C_VEL
LIN {X 0,Y 302.034,Z 535.694,A -85,B 0,C 180,E1 -16626.517,E2 -16626.517} C_VEL
LIN {X 0,Y 300.725,Z 548.153,A -85,B 0,C 180,E1 -16627.319,E2 -16627.319} C_VEL
LIN {X 0,Y 299.313,Z 559.267,A -85,B 0,C 180,E1 -16628.296,E2 -16628.296} C_VEL
LIN {X 0,Y 297.615,Z 570.85,A -85,B 0,C 180,E1 -16629.616,E2 -16629.616} C_VEL
LIN {X 0,Y 295.852,Z 581.282,A -85,B 0,C 180,E1 -16631.116,E2 -16631.116} C_VEL
LIN {X 0,Y 294.281,Z 590.63,A -85,B 0,C 180,E1 -16632.8,E2 -16632.8} C_VEL
LIN {X 0,Y 292.875,Z 599.08,A -85,B 0,C 180,E1 -16634.695,E2 -16634.695} C_VEL
LIN {X 0,Y 291.573,Z 606.525,A -85,B 0,C 180,E1 -16636.763,E2 -16636.763} C_VEL
LIN {X 0,Y 290.618,Z 612.51,A -85,B 0,C 180,E1 -16638.845,E2 -16638.845} C_VEL
LIN {X 0,Y 290.005,Z 617.244,A -85,B 0,C 180,E1 -16640.937,E2 -16640.937} C_VEL
LIN {X 0,Y 289.609,Z 620.864,A -85,B 0,C 180,E1 -16643.031,E2 -16643.031} C_VEL
LIN {X 0,Y 289.475,Z 622.828,A -85,B 0,C 180,E1 -16644.513,E2 -16644.513} C_VEL
LIN {X 0,Y 289.475,Z 625.139,A -85,B 0,C 180,E1 -16647.217,E2 -16647.217} C_VEL
LIN {X 0,Y 289.458,Z 625.749,A -85,B 0,C 180,E1 -16648.609,E2 -16648.609} C_VEL
LIN {X 0,Y 289.496,Z 625.965,A -85,B 0,C 180,E1 -16650,E2 -16650} C_VEL
LIN {X 0,Y 289.458,Z 625.742,A -85,B 0,C 180,E1 -16651.391,E2 -16651.391} C_VEL
LIN {X 0,Y 289.475,Z 625.127,A -85,B 0,C 180,E1 -16652.783,E2 -16652.783} C_VEL
LIN {X 0,Y 289.479,Z 622.798,A -85,B 0,C 180,E1 -16655.494,E2 -16655.494} C_VEL
LIN {X 0,Y 289.715,Z 619.752,A -85,B 0,C 180,E1 -16657.667,E2 -16657.667} C_VEL
LIN {X 0,Y 290.158,Z 615.754,A -85,B 0,C 180,E1 -16659.761,E2 -16659.761} C_VEL
LIN {X 0,Y 290.995,Z 609.613,A -85,B 0,C 180,E1 -16662.2,E2 -16662.2} C_VEL
LIN {X 0,Y 292.227,Z 602.918,A -85,B 0,C 180,E1 -16664.271,E2 -16664.271} C_VEL
LIN {X 0,Y 293.71,Z 594.615,A -85,B 0,C 180,E1 -16666.329,E2 -16666.329} C_VEL
LIN {X 0,Y 295.044,Z 586.098,A -85,B 0,C 180,E1 -16668.038,E2 -16668.038} C_VEL
LIN {X 0,Y 296.808,Z 575.587,A -85,B 0,C 180,E1 -16669.719,E2 -16669.719} C_VEL
LIN {X 0,Y 298.659,Z 563.762,A -85,B 0,C 180,E1 -16671.21,E2 -16671.21} C_VEL
LIN {X 0,Y 300.232,Z 551.856,A -85,B 0,C 180,E1 -16672.357,E2 -16672.357} C_VEL
LIN {X 0,Y 301.585,Z 539.467,A -85,B 0,C 180,E1 -16673.247,E2 -16673.247} C_VEL
LIN {X 0,Y 302.711,Z 526.723,A -85,B 0,C 180,E1 -16673.881,E2 -16673.881} C_VEL
LIN {X 0,Y 303.321,Z 513.266,A -85,B 0,C 180,E1 -16674.284,E2 -16674.284} C_VEL
LIN {X 0,Y 304.546,Z 457.464,A -85,B 0,C 180,E1 -16675.599,E2 -16675.599} C_VEL
LIN {X 0,Y 300.299,Z 429.574,A -85,B 0,C 180,E1 -16676.71,E2 -16676.71} C_VEL
LIN {X 0,Y 297.767,Z 416.916,A -85,B 0,C 180,E1 -16677.288,E2 -16677.288} C_VEL
LIN {X 0,Y 296.35,Z 412.977,A -85,B 0,C 180,E1 -16677.555,E2 -16677.555} C_VEL
LIN {X 0,Y 294.389,Z 403.192,A -85,B 0,C 180,E1 -16680.747,E2 -16680.747} C_VEL
LIN {X 0,Y 291.9,Z 392.493,A -85,B 0,C 180,E1 -16684.434,E2 -16684.434} C_VEL
LIN {X 0,Y 291.401,Z 390.191,A -85,B 0,C 180,E1 -16685.296,E2 -16685.296} C_VEL
LIN {X 0,Y 291.369,Z 390.19,A -85,B 0,C 180,E1 -16688.838,E2 -16688.838} C_VEL
LIN {X 0,Y 291.346,Z 390.191,A -85,B 0,C 180,E1 -16692.486,E2 -16692.486} C_VEL
LIN {X 0,Y 291.368,Z 390.185,A -85,B 0,C 180,E1 -16696.353,E2 -16696.353} C_VEL
LIN {X 0,Y 291.4,Z 390.185,A -85,B 0,C 180,E1 -16700.512,E2 -16700.512} C_VEL
LIN {X 0,Y 291.425,Z 390.181,A -85,B 0,C 180,E1 -16702.922,E2 -16702.922} C_VEL
LIN {X 0,Y 291.34,Z 390.189,A -85,B 0,C 180,E1 -16706.301,E2 -16706.301} C_VEL
LIN {X 0,Y 291.382,Z 390.185,A -85,B 0,C 180,E1 -16710.26,E2 -16710.26} C_VEL
LIN {X 0,Y 291.415,Z 390.182,A -85,B 0,C 180,E1 -16714.272,E2 -16714.272} C_VEL
LIN {X 0,Y 291.376,Z 390.185,A -85,B 0,C 180,E1 -16717.299,E2 -16717.299} C_VEL
LIN {X 0,Y 291.453,Z 390.177,A -85,B 0,C 180,E1 -16720.27,E2 -16720.27} C_VEL
LIN {X 0,Y 291.535,Z 390.166,A -85,B 0,C 180,E1 -16724.634,E2 -16724.634} C_VEL
LIN {X 0,Y 291.532,Z 390.166,A -85,B 0,C 180,E1 -16728.88,E2 -16728.88} C_VEL
LIN {X 0,Y 291.702,Z 390.147,A -85,B 0,C 180,E1 -16731.688,E2 -16731.688} C_VEL
LIN {X 0,Y 291.625,Z 390.158,A -85,B 0,C 180,E1 -16734.468,E2 -16734.468} C_VEL
LIN {X 0,Y 291.885,Z 390.121,A -85,B 0,C 180,E1 -16738.62,E2 -16738.62} C_VEL
LIN {X 0,Y 291.885,Z 390.125,A -85,B 0,C 180,E1 -16741.38,E2 -16741.38} C_VEL
LIN {X 0,Y 291.74,Z 390.144,A -85,B 0,C 180,E1 -16746.918,E2 -16746.918} C_VEL
LIN {X 0,Y 291.624,Z 390.156,A -85,B 0,C 180,E1 -16749.712,E2 -16749.712} C_VEL
LIN {X 0,Y 291.517,Z 390.167,A -85,B 0,C 180,E1 -16753.951,E2 -16753.951} C_VEL
LIN {X 0,Y 291.481,Z 390.177,A -85,B 0,C 180,E1 -16756.818,E2 -16756.818} C_VEL
LIN {X 0,Y 291.446,Z 390.172,A -85,B 0,C 180,E1 -16759.875,E2 -16759.875} C_VEL
LIN {X 0,Y 291.395,Z 390.187,A -85,B 0,C 180,E1 -16764.206,E2 -16764.206} C_VEL
LIN {X 0,Y 291.418,Z 390.182,A -85,B 0,C 180,E1 -16767.272,E2 -16767.272} C_VEL
LIN {X 0,Y 291.333,Z 390.194,A -85,B 0,C 180,E1 -16770.438,E2 -16770.438} C_VEL
LIN {X 0,Y 291.341,Z 390.192,A -85,B 0,C 180,E1 -16773.699,E2 -16773.699} C_VEL
LIN {X 0,Y 291.401,Z 390.183,A -85,B 0,C 180,E1 -16777.262,E2 -16777.262} C_VEL
LIN {X 0,Y 291.398,Z 390.184,A -85,B 0,C 180,E1 -16780.632,E2 -16780.632} C_VEL
LIN {X 0,Y 291.351,Z 390.192,A -85,B 0,C 180,E1 -16784.391,E2 -16784.391} C_VEL
LIN {X 0,Y 291.33,Z 390.195,A -85,B 0,C 180,E1 -16788.404,E2 -16788.404} C_VEL
LIN {X 0,Y 291.363,Z 390.19,A -85,B 0,C 180,E1 -16791.161,E2 -16791.161} C_VEL
LIN {X 0,Y 291.385,Z 390.191,A -85,B 0,C 180,E1 -16794.63,E2 -16794.63} C_VEL
LIN {X 0,Y 291.371,Z 390.192,A -85,B 0,C 180,E1 -16797.951,E2 -16797.951} C_VEL
LIN {X 0,Y 291.428,Z 390.332,A -85,B 0,C 180,E1 -16800.644,E2 -16800.644} C_VEL
LIN {X 0,Y 292.35,Z 394.184,A -85,B 0,C 180,E1 -16802.126,E2 -16802.126} C_VEL
LIN {X 0,Y 300.143,Z 412.159,A -85,B 0,C 180,E1 -16803.392,E2 -16803.392} C_VEL
LIN {X 0,Y 305.316,Z 425.832,A -85,B 0,C 180,E1 -16804.235,E2 -16804.235} C_VEL
LIN {X 0,Y 304.544,Z 461.601,A -85,B 0,C 180,E1 -16805.081,E2 -16805.081} C_VEL
LIN {X 0,Y 303.455,Z 501.394,A -85,B 0,C 180,E1 -16806.045,E2 -16806.045} C_VEL
LIN {X 0,Y 302.555,Z 515.128,A -85,B 0,C 180,E1 -16806.651,E2 -16806.651} C_VEL
LIN {X 0,Y 301.543,Z 527.443,A -85,B 0,C 180,E1 -16807.474,E2 -16807.474} C_VEL
LIN {X 0,Y 300.177,Z 539.25,A -85,B 0,C 180,E1 -16808.542,E2 -16808.542} C_VEL
LIN {X 0,Y 298.597,Z 550.586,A -85,B 0,C 180,E1 -16809.866,E2 -16809.866} C_VEL
LIN {X 0,Y 297.287,Z 560.439,A -85,B 0,C 180,E1 -16811.329,E2 -16811.329} C_VEL
LIN {X 0,Y 295.6,Z 569.951,A -85,B 0,C 180,E1 -16813.068,E2 -16813.068} C_VEL
LIN {X 0,Y 293.881,Z 578.851,A -85,B 0,C 180,E1 -16815.103,E2 -16815.103} C_VEL
LIN {X 0,Y 292.589,Z 586.007,A -85,B 0,C 180,E1 -16817.163,E2 -16817.163} C_VEL
LIN {X 0,Y 291.677,Z 590.832,A -85,B 0,C 180,E1 -16818.886,E2 -16818.886} C_VEL
LIN {X 0,Y 290.798,Z 595.52,A -85,B 0,C 180,E1 -16820.962,E2 -16820.962} C_VEL
LIN {X 0,Y 290.227,Z 599.245,A -85,B 0,C 180,E1 -16823.14,E2 -16823.14} C_VEL
LIN {X 0,Y 289.999,Z 600.953,A -85,B 0,C 180,E1 -16824.437,E2 -16824.437} C_VEL
LIN {X 0,Y 289.807,Z 602.345,A -85,B 0,C 180,E1 -16825.828,E2 -16825.828} C_VEL
LIN {X 0,Y 289.517,Z 603.946,A -85,B 0,C 180,E1 -16828.609,E2 -16828.609} C_VEL
LIN {X 0,Y 289.504,Z 604.176,A -85,B 0,C 180,E1 -16830,E2 -16830} C_VEL
LIN {X 0,Y 289.517,Z 603.985,A -85,B 0,C 180,E1 -16831.391,E2 -16831.391} C_VEL
LIN {X 0,Y 289.806,Z 602.433,A -85,B 0,C 180,E1 -16834.172,E2 -16834.172} C_VEL
LIN {X 0,Y 290.001,Z 601.08,A -85,B 0,C 180,E1 -16835.563,E2 -16835.563} C_VEL
LIN {X 0,Y 290.442,Z 598.219,A -85,B 0,C 180,E1 -16837.648,E2 -16837.648} C_VEL
LIN {X 0,Y 291.027,Z 594.342,A -85,B 0,C 180,E1 -16839.732,E2 -16839.732} C_VEL
LIN {X 0,Y 291.985,Z 589.332,A -85,B 0,C 180,E1 -16841.805,E2 -16841.805} C_VEL
LIN {X 0,Y 293.172,Z 583.023,A -85,B 0,C 180,E1 -16843.87,E2 -16843.87} C_VEL
LIN {X 0,Y 294.618,Z 575.125,A -85,B 0,C 180,E1 -16845.922,E2 -16845.922} C_VEL
LIN {X 0,Y 296.133,Z 567.067,A -85,B 0,C 180,E1 -16847.613,E2 -16847.613} C_VEL
LIN {X 0,Y 297.662,Z 557.238,A -85,B 0,C 180,E1 -16849.302,E2 -16849.302} C_VEL
LIN {X 0,Y 299.285,Z 546.168,A -85,B 0,C 180,E1 -16850.804,E2 -16850.804} C_VEL
LIN {X 0,Y 300.696,Z 535.311,A -85,B 0,C 180,E1 -16851.959,E2 -16851.959} C_VEL
LIN {X 0,Y 302.039,Z 523.307,A -85,B 0,C 180,E1 -16852.938,E2 -16852.938} C_VEL
LIN {X 0,Y 302.958,Z 510.975,A -85,B 0,C 180,E1 -16853.679,E2 -16853.679} C_VEL
LIN {X 0,Y 303.65,Z 498.186,A -85,B 0,C 180,E1 -16854.165,E2 -16854.165} C_VEL
LIN {X 0,Y 305.376,Z 426.09,A -85,B 0,C 180,E1 -16855.87,E2 -16855.87} C_VEL
LIN {X 0,Y 299.185,Z 409.672,A -85,B 0,C 180,E1 -16856.886,E2 -16856.886} C_VEL
LIN {X 0,Y 292.332,Z 394.049,A -85,B 0,C 180,E1 -16858.02,E2 -16858.02} C_VEL
LIN {X 0,Y 291.395,Z 390.191,A -85,B 0,C 180,E1 -16859.603,E2 -16859.603} C_VEL
LIN {X 0,Y 291.344,Z 390.191,A -85,B 0,C 180,E1 -16863.697,E2 -16863.697} C_VEL
LIN {X 0,Y 291.393,Z 390.188,A -85,B 0,C 180,E1 -16867.258,E2 -16867.258} C_VEL
LIN {X 0,Y 291.333,Z 390.193,A -85,B 0,C 180,E1 -16870.641,E2 -16870.641} C_VEL
LIN {X 0,Y 291.34,Z 390.193,A -85,B 0,C 180,E1 -16874.391,E2 -16874.391} C_VEL
LIN {X 0,Y 291.384,Z 390.183,A -85,B 0,C 180,E1 -16878.39,E2 -16878.39} C_VEL
LIN {X 0,Y 291.382,Z 390.189,A -85,B 0,C 180,E1 -16881.163,E2 -16881.163} C_VEL
LIN {X 0,Y 291.382,Z 390.187,A -85,B 0,C 180,E1 -16884.629,E2 -16884.629} C_VEL
LIN {X 0,Y 291.368,Z 390.191,A -85,B 0,C 180,E1 -16887.95,E2 -16887.95} C_VEL
LIN {X 0,Y 291.374,Z 390.186,A -85,B 0,C 180,E1 -16890.528,E2 -16890.528} C_VEL
LIN {X 0,Y 290.696,Z 390.273,A -85,B 0,C 180,E1 -16891.681,E2 -16891.681} C_VEL
LIN {X 0,Y 287.847,Z 390.632,A -85,B 0,C 180,E1 -16893.559,E2 -16893.559} C_VEL
LIN {X 0,Y 285.448,Z 390.928,A -85,B 0,C 180,E1 -16895.084,E2 -16895.084} C_VEL
LIN {X 0,Y 284.435,Z 391.048,A -85,B 0,C 180,E1 -16896.265,E2 -16896.265} C_VEL
LIN {X 0,Y 284.36,Z 391.057,A -85,B 0,C 180,E1 -16896.665,E2 -16896.665} C_VEL
LIN {X 0,Y 284.398,Z 391.058,A -85,B 0,C 180,E1 -16901.261,E2 -16901.261} C_VEL
LIN {X 0,Y 284.473,Z 391.046,A -85,B 0,C 180,E1 -16904.469,E2 -16904.469} C_VEL
LIN {X 0,Y 284.484,Z 391.042,A -85,B 0,C 180,E1 -16908.601,E2 -16908.601} C_VEL
LIN {X 0,Y 284.653,Z 391.028,A -85,B 0,C 180,E1 -16911.481,E2 -16911.481} C_VEL
LIN {X 0,Y 284.596,Z 391.03,A -85,B 0,C 180,E1 -16914.331,E2 -16914.331} C_VEL
LIN {X 0,Y 284.851,Z 391.001,A -85,B 0,C 180,E1 -16918.586,E2 -16918.586} C_VEL
LIN {X 0,Y 284.851,Z 390.995,A -85,B 0,C 180,E1 -16921.414,E2 -16921.414} C_VEL
LIN {X 0,Y 284.692,Z 391.019,A -85,B 0,C 180,E1 -16927.09,E2 -16927.09} C_VEL
LIN {X 0,Y 284.561,Z 391.034,A -85,B 0,C 180,E1 -16929.955,E2 -16929.955} C_VEL
LIN {X 0,Y 284.476,Z 391.043,A -85,B 0,C 180,E1 -16934.303,E2 -16934.303} C_VEL
LIN {X 0,Y 284.419,Z 391.056,A -85,B 0,C 180,E1 -16937.249,E2 -16937.249} C_VEL
LIN {X 0,Y 284.373,Z 391.056,A -85,B 0,C 180,E1 -16940.243,E2 -16940.243} C_VEL
LIN {X 0,Y 284.364,Z 391.06,A -85,B 0,C 180,E1 -16943.876,E2 -16943.876} C_VEL
LIN {X 0,Y 284.394,Z 391.059,A -85,B 0,C 180,E1 -16947.175,E2 -16947.175} C_VEL
LIN {X 0,Y 284.291,Z 391.07,A -85,B 0,C 180,E1 -16951.275,E2 -16951.275} C_VEL
LIN {X 0,Y 284.358,Z 391.061,A -85,B 0,C 180,E1 -16955.354,E2 -16955.354} C_VEL
LIN {X 0,Y 284.328,Z 391.064,A -85,B 0,C 180,E1 -16958.167,E2 -16958.167} C_VEL
LIN {X 0,Y 284.338,Z 391.065,A -85,B 0,C 180,E1 -16962.141,E2 -16962.141} C_VEL
LIN {X 0,Y 284.294,Z 391.071,A -85,B 0,C 180,E1 -16966.198,E2 -16966.198} C_VEL
LIN {X 0,Y 284.349,Z 391.067,A -85,B 0,C 180,E1 -16970.014,E2 -16970.014} C_VEL
LIN {X 0,Y 284.363,Z 391.151,A -85,B 0,C 180,E1 -16974.125,E2 -16974.125} C_VEL
LIN {X 0,Y 286.698,Z 401.271,A -85,B 0,C 180,E1 -16977.781,E2 -16977.781} C_VEL
LIN {X 0,Y 288.807,Z 411.184,A -85,B 0,C 180,E1 -16981.169,E2 -16981.169} C_VEL
LIN {X 0,Y 289.113,Z 412.717,A -85,B 0,C 180,E1 -16981.679,E2 -16981.679} C_VEL
LIN {X 0,Y 292.263,Z 421.292,A -85,B 0,C 180,E1 -16982.248,E2 -16982.248} C_VEL
LIN {X 0,Y 297.229,Z 451.035,A -85,B 0,C 180,E1 -16983.533,E2 -16983.533} C_VEL
LIN {X 0,Y 298.271,Z 460.52,A -85,B 0,C 180,E1 -16983.88,E2 -16983.88} C_VEL
LIN {X 0,Y 296.596,Z 521.511,A -85,B 0,C 180,E1 -16985.362,E2 -16985.362} C_VEL
LIN {X 0,Y 295.526,Z 535.436,A -85,B 0,C 180,E1 -16985.968,E2 -16985.968} C_VEL
LIN {X 0,Y 294.197,Z 547.892,A -85,B 0,C 180,E1 -16986.787,E2 -16986.787} C_VEL
LIN {X 0,Y 292.722,Z 559.004,A -85,B 0,C 180,E1 -16987.782,E2 -16987.782} C_VEL
LIN {X 0,Y 290.96,Z 570.586,A -85,B 0,C 180,E1 -16989.129,E2 -16989.129} C_VEL
LIN {X 0,Y 289.102,Z 581.016,A -85,B 0,C 180,E1 -16990.658,E2 -16990.658} C_VEL
LIN {X 0,Y 287.582,Z 589.694,A -85,B 0,C 180,E1 -16992.243,E2 -16992.243} C_VEL
LIN {X 0,Y 286.272,Z 597.436,A -85,B 0,C 180,E1 -16993.968,E2 -16993.968} C_VEL
LIN {X 0,Y 284.849,Z 605.135,A -85,B 0,C 180,E1 -16996.081,E2 -16996.081} C_VEL
LIN {X 0,Y 283.593,Z 612.242,A -85,B 0,C 180,E1 -16998.565,E2 -16998.565} C_VEL
LIN {X 0,Y 282.952,Z 616.977,A -85,B 0,C 180,E1 -17000.709,E2 -17000.709} C_VEL
LIN {X 0,Y 282.555,Z 620.597,A -85,B 0,C 180,E1 -17002.856,E2 -17002.856} C_VEL
LIN {X 0,Y 282.37,Z 622.8,A -85,B 0,C 180,E1 -17004.608,E2 -17004.608} C_VEL
LIN {X 0,Y 282.379,Z 624.872,A -85,B 0,C 180,E1 -17007.147,E2 -17007.147} C_VEL
LIN {X 0,Y 282.379,Z 625.483,A -85,B 0,C 180,E1 -17008.574,E2 -17008.574} C_VEL
LIN {X 0,Y 282.413,Z 625.698,A -85,B 0,C 180,E1 -17010,E2 -17010} C_VEL
LIN {X 0,Y 282.379,Z 625.475,A -85,B 0,C 180,E1 -17011.426,E2 -17011.426} C_VEL
LIN {X 0,Y 282.378,Z 624.86,A -85,B 0,C 180,E1 -17012.853,E2 -17012.853} C_VEL
LIN {X 0,Y 282.402,Z 622.708,A -85,B 0,C 180,E1 -17015.46,E2 -17015.46} C_VEL
LIN {X 0,Y 282.67,Z 619.484,A -85,B 0,C 180,E1 -17017.859,E2 -17017.859} C_VEL
LIN {X 0,Y 283.132,Z 615.485,A -85,B 0,C 180,E1 -17020.006,E2 -17020.006} C_VEL
LIN {X 0,Y 284.031,Z 609.343,A -85,B 0,C 180,E1 -17022.504,E2 -17022.504} C_VEL
LIN {X 0,Y 285.338,Z 602.649,A -85,B 0,C 180,E1 -17024.623,E2 -17024.623} C_VEL
LIN {X 0,Y 286.878,Z 594.344,A -85,B 0,C 180,E1 -17026.729,E2 -17026.729} C_VEL
LIN {X 0,Y 288.272,Z 585.826,A -85,B 0,C 180,E1 -17028.477,E2 -17028.477} C_VEL
LIN {X 0,Y 290.138,Z 575.317,A -85,B 0,C 180,E1 -17030.192,E2 -17030.192} C_VEL
LIN {X 0,Y 292.059,Z 563.49,A -85,B 0,C 180,E1 -17031.714,E2 -17031.714} C_VEL
LIN {X 0,Y 293.66,Z 551.582,A -85,B 0,C 180,E1 -17032.886,E2 -17032.886} C_VEL
LIN {X 0,Y 295.083,Z 539.193,A -85,B 0,C 180,E1 -17033.79,E2 -17033.79} C_VEL
LIN {X 0,Y 296.216,Z 526.443,A -85,B 0,C 180,E1 -17034.438,E2 -17034.438} C_VEL
LIN {X 0,Y 296.865,Z 512.977,A -85,B 0,C 180,E1 -17034.848,E2 -17034.848} C_VEL
LIN {X 0,Y 298.146,Z 458.492,A -85,B 0,C 180,E1 -17036.155,E2 -17036.155} C_VEL
LIN {X 0,Y 294.041,Z 431.284,A -85,B 0,C 180,E1 -17037.272,E2 -17037.272} C_VEL
LIN {X 0,Y 291.676,Z 419.32,A -85,B 0,C 180,E1 -17037.834,E2 -17037.834} C_VEL
LIN {X 0,Y 289.13,Z 412.658,A -85,B 0,C 180,E1 -17038.31,E2 -17038.31} C_VEL
LIN {X 0,Y 287.376,Z 404.293,A -85,B 0,C 180,E1 -17041.135,E2 -17041.135} C_VEL
LIN {X 0,Y 285.168,Z 394.696,A -85,B 0,C 180,E1 -17044.529,E2 -17044.529} C_VEL
LIN {X 0,Y 284.347,Z 391.069,A -85,B 0,C 180,E1 -17045.946,E2 -17045.946} C_VEL
LIN {X 0,Y 284.349,Z 391.066,A -85,B 0,C 180,E1 -17049.986,E2 -17049.986} C_VEL
LIN {X 0,Y 284.291,Z 391.065,A -85,B 0,C 180,E1 -17054.2,E2 -17054.2} C_VEL
LIN {X 0,Y 284.335,Z 391.065,A -85,B 0,C 180,E1 -17058.136,E2 -17058.136} C_VEL
LIN {X 0,Y 284.337,Z 391.063,A -85,B 0,C 180,E1 -17062.272,E2 -17062.272} C_VEL
LIN {X 0,Y 284.32,Z 391.07,A -85,B 0,C 180,E1 -17065.352,E2 -17065.352} C_VEL
LIN {X 0,Y 284.291,Z 391.07,A -85,B 0,C 180,E1 -17068.725,E2 -17068.725} C_VEL
LIN {X 0,Y 284.395,Z 391.055,A -85,B 0,C 180,E1 -17072.825,E2 -17072.825} C_VEL
LIN {X 0,Y 284.361,Z 391.056,A -85,B 0,C 180,E1 -17076.706,E2 -17076.706} C_VEL
LIN {X 0,Y 284.398,Z 391.056,A -85,B 0,C 180,E1 -17081.261,E2 -17081.261} C_VEL
LIN {X 0,Y 284.472,Z 391.045,A -85,B 0,C 180,E1 -17084.469,E2 -17084.469} C_VEL
LIN {X 0,Y 284.484,Z 391.045,A -85,B 0,C 180,E1 -17088.601,E2 -17088.601} C_VEL
LIN {X 0,Y 284.653,Z 391.026,A -85,B 0,C 180,E1 -17091.481,E2 -17091.481} C_VEL
LIN {X 0,Y 284.596,Z 391.033,A -85,B 0,C 180,E1 -17094.331,E2 -17094.331} C_VEL
LIN {X 0,Y 284.851,Z 390.996,A -85,B 0,C 180,E1 -17098.586,E2 -17098.586} C_VEL
LIN {X 0,Y 284.851,Z 391.001,A -85,B 0,C 180,E1 -17101.414,E2 -17101.414} C_VEL
LIN {X 0,Y 284.692,Z 391.023,A -85,B 0,C 180,E1 -17107.09,E2 -17107.09} C_VEL
LIN {X 0,Y 284.561,Z 391.036,A -85,B 0,C 180,E1 -17109.956,E2 -17109.956} C_VEL
LIN {X 0,Y 284.473,Z 391.046,A -85,B 0,C 180,E1 -17114.303,E2 -17114.303} C_VEL
LIN {X 0,Y 284.42,Z 391.053,A -85,B 0,C 180,E1 -17117.249,E2 -17117.249} C_VEL
LIN {X 0,Y 284.374,Z 391.054,A -85,B 0,C 180,E1 -17120.243,E2 -17120.243} C_VEL
LIN {X 0,Y 284.364,Z 391.061,A -85,B 0,C 180,E1 -17123.876,E2 -17123.876} C_VEL
LIN {X 0,Y 284.393,Z 391.057,A -85,B 0,C 180,E1 -17127.174,E2 -17127.174} C_VEL
LIN {X 0,Y 284.291,Z 391.065,A -85,B 0,C 180,E1 -17131.275,E2 -17131.275} C_VEL
LIN {X 0,Y 284.359,Z 391.061,A -85,B 0,C 180,E1 -17135.355,E2 -17135.355} C_VEL
LIN {X 0,Y 284.333,Z 391.066,A -85,B 0,C 180,E1 -17138.166,E2 -17138.166} C_VEL
LIN {X 0,Y 284.338,Z 391.065,A -85,B 0,C 180,E1 -17142.141,E2 -17142.141} C_VEL
LIN {X 0,Y 284.295,Z 391.073,A -85,B 0,C 180,E1 -17146.198,E2 -17146.198} C_VEL
LIN {X 0,Y 284.306,Z 391.073,A -85,B 0,C 180,E1 -17150.025,E2 -17150.025} C_VEL
LIN {X 0,Y 284.349,Z 391.065,A -85,B 0,C 180,E1 -17153.618,E2 -17153.618} C_VEL
LIN {X 0,Y 284.307,Z 391.071,A -85,B 0,C 180,E1 -17157.19,E2 -17157.19} C_VEL
LIN {X 0,Y 284.328,Z 391.147,A -85,B 0,C 180,E1 -17160.034,E2 -17160.034} C_VEL
LIN {X 0,Y 285.14,Z 394.398,A -85,B 0,C 180,E1 -17161.353,E2 -17161.353} C_VEL
LIN {X 0,Y 293.365,Z 412.865,A -85,B 0,C 180,E1 -17162.738,E2 -17162.738} C_VEL
LIN {X 0,Y 298.989,Z 427.428,A -85,B 0,C 180,E1 -17163.683,E2 -17163.683} C_VEL
LIN {X 0,Y 297.07,Z 500.524,A -85,B 0,C 180,E1 -17165.451,E2 -17165.451} C_VEL
LIN {X 0,Y 296.172,Z 513.884,A -85,B 0,C 180,E1 -17166.024,E2 -17166.024} C_VEL
LIN {X 0,Y 295.149,Z 526.624,A -85,B 0,C 180,E1 -17166.866,E2 -17166.866} C_VEL
LIN {X 0,Y 293.808,Z 537.94,A -85,B 0,C 180,E1 -17167.868,E2 -17167.868} C_VEL
LIN {X 0,Y 292.165,Z 549.57,A -85,B 0,C 180,E1 -17169.219,E2 -17169.219} C_VEL
LIN {X 0,Y 290.691,Z 559.882,A -85,B 0,C 180,E1 -17170.747,E2 -17170.747} C_VEL
LIN {X 0,Y 289.104,Z 568.533,A -85,B 0,C 180,E1 -17172.31,E2 -17172.31} C_VEL
LIN {X 0,Y 287.624,Z 576.387,A -85,B 0,C 180,E1 -17174.045,E2 -17174.045} C_VEL
LIN {X 0,Y 286.109,Z 584.06,A -85,B 0,C 180,E1 -17176.143,E2 -17176.143} C_VEL
LIN {X 0,Y 284.7,Z 591.101,A -85,B 0,C 180,E1 -17178.61,E2 -17178.61} C_VEL
LIN {X 0,Y 283.791,Z 595.788,A -85,B 0,C 180,E1 -17180.737,E2 -17180.737} C_VEL
LIN {X 0,Y 283.15,Z 599.764,A -85,B 0,C 180,E1 -17183.138,E2 -17183.138} C_VEL
LIN {X 0,Y 282.751,Z 602.611,A -85,B 0,C 180,E1 -17185.724,E2 -17185.724} C_VEL
LIN {X 0,Y 282.438,Z 604.213,A -85,B 0,C 180,E1 -17188.574,E2 -17188.574} C_VEL
LIN {X 0,Y 282.422,Z 604.443,A -85,B 0,C 180,E1 -17190,E2 -17190} C_VEL
LIN {X 0,Y 282.438,Z 604.251,A -85,B 0,C 180,E1 -17191.426,E2 -17191.426} C_VEL
LIN {X 0,Y 282.751,Z 602.699,A -85,B 0,C 180,E1 -17194.276,E2 -17194.276} C_VEL
LIN {X 0,Y 283.184,Z 599.843,A -85,B 0,C 180,E1 -17196.919,E2 -17196.919} C_VEL
LIN {X 0,Y 283.784,Z 596.018,A -85,B 0,C 180,E1 -17199.263,E2 -17199.263} C_VEL
LIN {X 0,Y 284.643,Z 591.394,A -85,B 0,C 180,E1 -17201.392,E2 -17201.392} C_VEL
LIN {X 0,Y 286.054,Z 584.418,A -85,B 0,C 180,E1 -17203.859,E2 -17203.859} C_VEL
LIN {X 0,Y 287.501,Z 576.857,A -85,B 0,C 180,E1 -17205.962,E2 -17205.962} C_VEL
LIN {X 0,Y 289.383,Z 567.33,A -85,B 0,C 180,E1 -17208.038,E2 -17208.038} C_VEL
LIN {X 0,Y 290.978,Z 557.501,A -85,B 0,C 180,E1 -17209.763,E2 -17209.763} C_VEL
LIN {X 0,Y 292.666,Z 546.43,A -85,B 0,C 180,E1 -17211.297,E2 -17211.297} C_VEL
LIN {X 0,Y 294.153,Z 535.571,A -85,B 0,C 180,E1 -17212.474,E2 -17212.474} C_VEL
LIN {X 0,Y 295.536,Z 523.565,A -85,B 0,C 180,E1 -17213.473,E2 -17213.473} C_VEL
LIN {X 0,Y 296.496,Z 511.229,A -85,B 0,C 180,E1 -17214.227,E2 -17214.227} C_VEL
LIN {X 0,Y 297.201,Z 498.432,A -85,B 0,C 180,E1 -17214.724,E2 -17214.724} C_VEL
LIN {X 0,Y 298.982,Z 427.422,A -85,B 0,C 180,E1 -17216.438,E2 -17216.438} C_VEL
LIN {X 0,Y 292.111,Z 409.802,A -85,B 0,C 180,E1 -17217.596,E2 -17217.596} C_VEL
LIN {X 0,Y 285.157,Z 394.368,A -85,B 0,C 180,E1 -17218.782,E2 -17218.782} C_VEL
LIN {X 0,Y 284.311,Z 391.069,A -85,B 0,C 180,E1 -17220.202,E2 -17220.202} C_VEL
LIN {X 0,Y 284.323,Z 391.069,A -85,B 0,C 180,E1 -17224.646,E2 -17224.646} C_VEL
LIN {X 0,Y 284.322,Z 391.069,A -85,B 0,C 180,E1 -17228.166,E2 -17228.166} C_VEL
LIN {X 0,Y 284.281,Z 391.072,A -85,B 0,C 180,E1 -17232.127,E2 -17232.127} C_VEL
LIN {X 0,Y 284.315,Z 391.06,A -85,B 0,C 180,E1 -17236.201,E2 -17236.201} C_VEL
LIN {X 0,Y 284.349,Z 391.066,A -85,B 0,C 180,E1 -17240.012,E2 -17240.012} C_VEL
LIN {X 0,Y 284.352,Z 391.064,A -85,B 0,C 180,E1 -17243.617,E2 -17243.617} C_VEL
LIN {X 0,Y 284.304,Z 391.067,A -85,B 0,C 180,E1 -17247.189,E2 -17247.189} C_VEL
LIN {X 0,Y 284.344,Z 391.061,A -85,B 0,C 180,E1 -17250.507,E2 -17250.507} C_VEL
LIN {X 0,Y 284.373,Z 391.064,A -85,B 0,C 180,E1 -17253.586,E2 -17253.586} C_VEL
LIN {X 0,Y 284.36,Z 391.057,A -85,B 0,C 180,E1 -17256.665,E2 -17256.665} C_VEL
LIN {X 0,Y 283.711,Z 391.143,A -85,B 0,C 180,E1 -17257.848,E2 -17257.848} C_VEL
LIN {X 0,Y 280.863,Z 391.499,A -85,B 0,C 180,E1 -17259.776,E2 -17259.776} C_VEL
LIN {X 0,Y 278.446,Z 391.798,A -85,B 0,C 180,E1 -17261.341,E2 -17261.341} C_VEL
LIN {X 0,Y 277.424,Z 391.92,A -85,B 0,C 180,E1 -17262.554,E2 -17262.554} C_VEL
LIN {X 0,Y 277.349,Z 391.929,A -85,B 0,C 180,E1 -17262.965,E2 -17262.965} C_VEL
LIN {X 0,Y 277.423,Z 391.93,A -85,B 0,C 180,E1 -17265.325,E2 -17265.325} C_VEL
LIN {X 0,Y 277.502,Z 391.914,A -85,B 0,C 180,E1 -17269.788,E2 -17269.788} C_VEL
LIN {X 0,Y 277.647,Z 391.9,A -85,B 0,C 180,E1 -17272.729,E2 -17272.729} C_VEL
LIN {X 0,Y 277.816,Z 391.878,A -85,B 0,C 180,E1 -17278.55,E2 -17278.55} C_VEL
LIN {X 0,Y 277.817,Z 391.87,A -85,B 0,C 180,E1 -17281.45,E2 -17281.45} C_VEL
LIN {X 0,Y 277.647,Z 391.894,A -85,B 0,C 180,E1 -17287.271,E2 -17287.271} C_VEL
LIN {X 0,Y 277.501,Z 391.914,A -85,B 0,C 180,E1 -17290.211,E2 -17290.211} C_VEL
LIN {X 0,Y 277.429,Z 391.921,A -85,B 0,C 180,E1 -17294.674,E2 -17294.674} C_VEL
LIN {X 0,Y 277.34,Z 391.932,A -85,B 0,C 180,E1 -17299.234,E2 -17299.234} C_VEL
LIN {X 0,Y 277.314,Z 391.939,A -85,B 0,C 180,E1 -17304.171,E2 -17304.171} C_VEL
LIN {X 0,Y 277.323,Z 391.938,A -85,B 0,C 180,E1 -17307.506,E2 -17307.506} C_VEL
LIN {X 0,Y 277.268,Z 391.947,A -85,B 0,C 180,E1 -17310.482,E2 -17310.482} C_VEL
LIN {X 0,Y 277.25,Z 391.943,A -85,B 0,C 180,E1 -17313.895,E2 -17313.895} C_VEL
LIN {X 0,Y 277.282,Z 391.939,A -85,B 0,C 180,E1 -17317.467,E2 -17317.467} C_VEL
LIN {X 0,Y 277.261,Z 391.945,A -85,B 0,C 180,E1 -17321.227,E2 -17321.227} C_VEL
LIN {X 0,Y 277.24,Z 391.949,A -85,B 0,C 180,E1 -17325.218,E2 -17325.218} C_VEL
LIN {X 0,Y 277.259,Z 391.948,A -85,B 0,C 180,E1 -17329.503,E2 -17329.503} C_VEL
LIN {X 0,Y 277.313,Z 392.034,A -85,B 0,C 180,E1 -17333.48,E2 -17333.48} C_VEL
LIN {X 0,Y 279.726,Z 402.263,A -85,B 0,C 180,E1 -17337.305,E2 -17337.305} C_VEL
LIN {X 0,Y 281.853,Z 412.444,A -85,B 0,C 180,E1 -17340.888,E2 -17340.888} C_VEL
LIN {X 0,Y 286.171,Z 423.508,A -85,B 0,C 180,E1 -17341.673,E2 -17341.673} C_VEL
LIN {X 0,Y 290.896,Z 452.202,A -85,B 0,C 180,E1 -17342.948,E2 -17342.948} C_VEL
LIN {X 0,Y 291.918,Z 460.307,A -85,B 0,C 180,E1 -17343.268,E2 -17343.268} C_VEL
LIN {X 0,Y 290.158,Z 521.258,A -85,B 0,C 180,E1 -17344.778,E2 -17344.778} C_VEL
LIN {X 0,Y 289.068,Z 535.178,A -85,B 0,C 180,E1 -17345.396,E2 -17345.396} C_VEL
LIN {X 0,Y 287.694,Z 547.631,A -85,B 0,C 180,E1 -17346.23,E2 -17346.23} C_VEL
LIN {X 0,Y 285.92,Z 560.327,A -85,B 0,C 180,E1 -17347.415,E2 -17347.415} C_VEL
LIN {X 0,Y 284.112,Z 571.618,A -85,B 0,C 180,E1 -17348.791,E2 -17348.791} C_VEL
LIN {X 0,Y 282.206,Z 581.791,A -85,B 0,C 180,E1 -17350.355,E2 -17350.355} C_VEL
LIN {X 0,Y 280.411,Z 591.532,A -85,B 0,C 180,E1 -17352.252,E2 -17352.252} C_VEL
LIN {X 0,Y 278.872,Z 599.909,A -85,B 0,C 180,E1 -17354.282,E2 -17354.282} C_VEL
LIN {X 0,Y 277.498,Z 607.11,A -85,B 0,C 180,E1 -17356.452,E2 -17356.452} C_VEL
LIN {X 0,Y 276.581,Z 611.974,A -85,B 0,C 180,E1 -17358.271,E2 -17358.271} C_VEL
LIN {X 0,Y 275.919,Z 616.709,A -85,B 0,C 180,E1 -17360.47,E2 -17360.47} C_VEL
LIN {X 0,Y 275.493,Z 620.33,A -85,B 0,C 180,E1 -17362.672,E2 -17362.672} C_VEL
LIN {X 0,Y 275.264,Z 622.776,A -85,B 0,C 180,E1 -17364.712,E2 -17364.712} C_VEL
LIN {X 0,Y 275.285,Z 624.605,A -85,B 0,C 180,E1 -17367.073,E2 -17367.073} C_VEL
LIN {X 0,Y 275.302,Z 625.217,A -85,B 0,C 180,E1 -17368.537,E2 -17368.537} C_VEL
LIN {X 0,Y 275.332,Z 625.432,A -85,B 0,C 180,E1 -17370,E2 -17370} C_VEL
LIN {X 0,Y 275.302,Z 625.209,A -85,B 0,C 180,E1 -17371.463,E2 -17371.463} C_VEL
LIN {X 0,Y 275.285,Z 624.592,A -85,B 0,C 180,E1 -17372.927,E2 -17372.927} C_VEL
LIN {X 0,Y 275.321,Z 622.628,A -85,B 0,C 180,E1 -17375.413,E2 -17375.413} C_VEL
LIN {X 0,Y 275.598,Z 619.214,A -85,B 0,C 180,E1 -17378.062,E2 -17378.062} C_VEL
LIN {X 0,Y 276.122,Z 615.216,A -85,B 0,C 180,E1 -17380.263,E2 -17380.263} C_VEL
LIN {X 0,Y 277.052,Z 609.072,A -85,B 0,C 180,E1 -17382.824,E2 -17382.824} C_VEL
LIN {X 0,Y 278.455,Z 602.379,A -85,B 0,C 180,E1 -17384.993,E2 -17384.993} C_VEL
LIN {X 0,Y 280.044,Z 594.073,A -85,B 0,C 180,E1 -17387.15,E2 -17387.15} C_VEL
LIN {X 0,Y 281.51,Z 585.555,A -85,B 0,C 180,E1 -17388.938,E2 -17388.938} C_VEL
LIN {X 0,Y 283.251,Z 576.222,A -85,B 0,C 180,E1 -17390.515,E2 -17390.515} C_VEL
LIN {X 0,Y 285.211,Z 564.649,A -85,B 0,C 180,E1 -17392.072,E2 -17392.072} C_VEL
LIN {X 0,Y 286.892,Z 553.249,A -85,B 0,C 180,E1 -17393.266,E2 -17393.266} C_VEL
LIN {X 0,Y 288.353,Z 541.523,A -85,B 0,C 180,E1 -17394.19,E2 -17394.19} C_VEL
LIN {X 0,Y 289.581,Z 528.922,A -85,B 0,C 180,E1 -17394.892,E2 -17394.892} C_VEL
LIN {X 0,Y 290.332,Z 516.07,A -85,B 0,C 180,E1 -17395.35,E2 -17395.35} C_VEL
LIN {X 0,Y 291.788,Z 459.567,A -85,B 0,C 180,E1 -17396.733,E2 -17396.733} C_VEL
LIN {X 0,Y 287.814,Z 432.956,A -85,B 0,C 180,E1 -17397.859,E2 -17397.859} C_VEL
LIN {X 0,Y 285.681,Z 422.053,A -85,B 0,C 180,E1 -17398.387,E2 -17398.387} C_VEL
LIN {X 0,Y 281.879,Z 412.352,A -85,B 0,C 180,E1 -17399.107,E2 -17399.107} C_VEL
LIN {X 0,Y 279.701,Z 402.149,A -85,B 0,C 180,E1 -17402.698,E2 -17402.698} C_VEL
LIN {X 0,Y 277.3,Z 391.945,A -85,B 0,C 180,E1 -17406.573,E2 -17406.573} C_VEL
LIN {X 0,Y 277.259,Z 391.948,A -85,B 0,C 180,E1 -17410.497,E2 -17410.497} C_VEL
LIN {X 0,Y 277.24,Z 391.939,A -85,B 0,C 180,E1 -17414.781,E2 -17414.781} C_VEL
LIN {X 0,Y 277.261,Z 391.946,A -85,B 0,C 180,E1 -17418.773,E2 -17418.773} C_VEL
LIN {X 0,Y 277.282,Z 391.942,A -85,B 0,C 180,E1 -17422.533,E2 -17422.533} C_VEL
LIN {X 0,Y 277.25,Z 391.945,A -85,B 0,C 180,E1 -17426.105,E2 -17426.105} C_VEL
LIN {X 0,Y 277.257,Z 391.947,A -85,B 0,C 180,E1 -17429.538,E2 -17429.538} C_VEL
LIN {X 0,Y 277.356,Z 391.932,A -85,B 0,C 180,E1 -17432.864,E2 -17432.864} C_VEL
LIN {X 0,Y 277.323,Z 391.932,A -85,B 0,C 180,E1 -17436.079,E2 -17436.079} C_VEL
LIN {X 0,Y 277.339,Z 391.937,A -85,B 0,C 180,E1 -17440.766,E2 -17440.766} C_VEL
LIN {X 0,Y 277.423,Z 391.929,A -85,B 0,C 180,E1 -17445.325,E2 -17445.325} C_VEL
LIN {X 0,Y 277.501,Z 391.908,A -85,B 0,C 180,E1 -17449.789,E2 -17449.789} C_VEL
LIN {X 0,Y 277.647,Z 391.899,A -85,B 0,C 180,E1 -17452.729,E2 -17452.729} C_VEL
LIN {X 0,Y 277.816,Z 391.872,A -85,B 0,C 180,E1 -17458.55,E2 -17458.55} C_VEL
LIN {X 0,Y 277.816,Z 391.877,A -85,B 0,C 180,E1 -17461.45,E2 -17461.45} C_VEL
LIN {X 0,Y 277.647,Z 391.899,A -85,B 0,C 180,E1 -17467.271,E2 -17467.271} C_VEL
LIN {X 0,Y 277.502,Z 391.916,A -85,B 0,C 180,E1 -17470.212,E2 -17470.212} C_VEL
LIN {X 0,Y 277.423,Z 391.926,A -85,B 0,C 180,E1 -17474.675,E2 -17474.675} C_VEL
LIN {X 0,Y 277.34,Z 391.928,A -85,B 0,C 180,E1 -17479.234,E2 -17479.234} C_VEL
LIN {X 0,Y 277.314,Z 391.941,A -85,B 0,C 180,E1 -17484.171,E2 -17484.171} C_VEL
LIN {X 0,Y 277.321,Z 391.937,A -85,B 0,C 180,E1 -17487.506,E2 -17487.506} C_VEL
LIN {X 0,Y 277.268,Z 391.945,A -85,B 0,C 180,E1 -17490.482,E2 -17490.482} C_VEL
LIN {X 0,Y 277.251,Z 391.948,A -85,B 0,C 180,E1 -17493.895,E2 -17493.895} C_VEL
LIN {X 0,Y 277.287,Z 391.94,A -85,B 0,C 180,E1 -17497.467,E2 -17497.467} C_VEL
LIN {X 0,Y 277.261,Z 391.943,A -85,B 0,C 180,E1 -17501.227,E2 -17501.227} C_VEL
LIN {X 0,Y 277.241,Z 391.947,A -85,B 0,C 180,E1 -17505.219,E2 -17505.219} C_VEL
LIN {X 0,Y 277.224,Z 391.953,A -85,B 0,C 180,E1 -17509.512,E2 -17509.512} C_VEL
LIN {X 0,Y 277.28,Z 391.947,A -85,B 0,C 180,E1 -17512.534,E2 -17512.534} C_VEL
LIN {X 0,Y 277.254,Z 391.951,A -85,B 0,C 180,E1 -17516.106,E2 -17516.106} C_VEL
LIN {X 0,Y 277.282,Z 392.09,A -85,B 0,C 180,E1 -17519.447,E2 -17519.447} C_VEL
LIN {X 0,Y 277.936,Z 394.739,A -85,B 0,C 180,E1 -17520.539,E2 -17520.539} C_VEL
LIN {X 0,Y 285.817,Z 411.832,A -85,B 0,C 180,E1 -17521.917,E2 -17521.917} C_VEL
LIN {X 0,Y 292.59,Z 429.124,A -85,B 0,C 180,E1 -17523.099,E2 -17523.099} C_VEL
LIN {X 0,Y 290.63,Z 500.808,A -85,B 0,C 180,E1 -17524.869,E2 -17524.869} C_VEL
LIN {X 0,Y 289.73,Z 514.161,A -85,B 0,C 180,E1 -17525.456,E2 -17525.456} C_VEL
LIN {X 0,Y 288.651,Z 526.898,A -85,B 0,C 180,E1 -17526.314,E2 -17526.314} C_VEL
LIN {X 0,Y 287.267,Z 538.212,A -85,B 0,C 180,E1 -17527.337,E2 -17527.337} C_VEL
LIN {X 0,Y 285.555,Z 549.841,A -85,B 0,C 180,E1 -17528.715,E2 -17528.715} C_VEL
LIN {X 0,Y 283.908,Z 560.719,A -85,B 0,C 180,E1 -17530.368,E2 -17530.368} C_VEL
LIN {X 0,Y 282.047,Z 570.491,A -85,B 0,C 180,E1 -17532.228,E2 -17532.228} C_VEL
LIN {X 0,Y 280.192,Z 579.389,A -85,B 0,C 180,E1 -17534.358,E2 -17534.358} C_VEL
LIN {X 0,Y 278.745,Z 586.546,A -85,B 0,C 180,E1 -17536.514,E2 -17536.514} C_VEL
LIN {X 0,Y 277.738,Z 591.37,A -85,B 0,C 180,E1 -17538.321,E2 -17538.321} C_VEL
LIN {X 0,Y 276.782,Z 596.057,A -85,B 0,C 180,E1 -17540.5,E2 -17540.5} C_VEL
LIN {X 0,Y 276.069,Z 600.27,A -85,B 0,C 180,E1 -17543.141,E2 -17543.141} C_VEL
LIN {X 0,Y 275.675,Z 602.879,A -85,B 0,C 180,E1 -17545.614,E2 -17545.614} C_VEL
LIN {X 0,Y 275.362,Z 604.479,A -85,B 0,C 180,E1 -17548.538,E2 -17548.538} C_VEL
LIN {X 0,Y 275.341,Z 604.709,A -85,B 0,C 180,E1 -17550,E2 -17550} C_VEL
LIN {X 0,Y 275.361,Z 604.517,A -85,B 0,C 180,E1 -17551.462,E2 -17551.462} C_VEL
LIN {X 0,Y 275.675,Z 602.965,A -85,B 0,C 180,E1 -17554.386,E2 -17554.386} C_VEL
LIN {X 0,Y 276.101,Z 600.342,A -85,B 0,C 180,E1 -17556.913,E2 -17556.913} C_VEL
LIN {X 0,Y 276.774,Z 596.284,A -85,B 0,C 180,E1 -17559.5,E2 -17559.5} C_VEL
LIN {X 0,Y 277.69,Z 591.66,A -85,B 0,C 180,E1 -17561.681,E2 -17561.681} C_VEL
LIN {X 0,Y 279.179,Z 584.683,A -85,B 0,C 180,E1 -17564.208,E2 -17564.208} C_VEL
LIN {X 0,Y 280.693,Z 577.122,A -85,B 0,C 180,E1 -17566.36,E2 -17566.36} C_VEL
LIN {X 0,Y 282.656,Z 567.594,A -85,B 0,C 180,E1 -17568.482,E2 -17568.482} C_VEL
LIN {X 0,Y 284.308,Z 557.765,A -85,B 0,C 180,E1 -17570.247,E2 -17570.247} C_VEL
LIN {X 0,Y 286.065,Z 546.693,A -85,B 0,C 180,E1 -17571.813,E2 -17571.813} C_VEL
LIN {X 0,Y 287.631,Z 535.831,A -85,B 0,C 180,E1 -17573.013,E2 -17573.013} C_VEL
LIN {X 0,Y 289.044,Z 523.825,A -85,B 0,C 180,E1 -17574.033,E2 -17574.033} C_VEL
LIN {X 0,Y 290.05,Z 511.484,A -85,B 0,C 180,E1 -17574.802,E2 -17574.802} C_VEL
LIN {X 0,Y 290.783,Z 498.678,A -85,B 0,C 180,E1 -17575.308,E2 -17575.308} C_VEL
LIN {X 0,Y 292.631,Z 429.157,A -85,B 0,C 180,E1 -17577.017,E2 -17577.017} C_VEL
LIN {X 0,Y 285.74,Z 411.585,A -85,B 0,C 180,E1 -17578.222,E2 -17578.222} C_VEL
LIN {X 0,Y 279.066,Z 397.328,A -85,B 0,C 180,E1 -17579.38,E2 -17579.38} C_VEL
LIN {X 0,Y 277.923,Z 394.598,A -85,B 0,C 180,E1 -17579.631,E2 -17579.631} C_VEL
LIN {X 0,Y 277.281,Z 391.943,A -85,B 0,C 180,E1 -17580.763,E2 -17580.763} C_VEL
LIN {X 0,Y 277.254,Z 391.946,A -85,B 0,C 180,E1 -17583.894,E2 -17583.894} C_VEL
LIN {X 0,Y 277.28,Z 391.947,A -85,B 0,C 180,E1 -17587.466,E2 -17587.466} C_VEL
LIN {X 0,Y 277.214,Z 391.953,A -85,B 0,C 180,E1 -17591.235,E2 -17591.235} C_VEL
LIN {X 0,Y 277.244,Z 391.95,A -85,B 0,C 180,E1 -17595.216,E2 -17595.216} C_VEL
LIN {X 0,Y 277.292,Z 391.941,A -85,B 0,C 180,E1 -17599.494,E2 -17599.494} C_VEL
LIN {X 0,Y 277.287,Z 391.939,A -85,B 0,C 180,E1 -17602.533,E2 -17602.533} C_VEL
LIN {X 0,Y 277.251,Z 391.945,A -85,B 0,C 180,E1 -17606.105,E2 -17606.105} C_VEL
LIN {X 0,Y 277.258,Z 391.95,A -85,B 0,C 180,E1 -17609.538,E2 -17609.538} C_VEL
LIN {X 0,Y 277.354,Z 391.933,A -85,B 0,C 180,E1 -17612.863,E2 -17612.863} C_VEL
LIN {X 0,Y 277.283,Z 391.937,A -85,B 0,C 180,E1 -17616.652,E2 -17616.652} C_VEL
LIN {X 0,Y 277.34,Z 391.937,A -85,B 0,C 180,E1 -17620.766,E2 -17620.766} C_VEL
LIN {X 0,Y 277.349,Z 391.929,A -85,B 0,C 180,E1 -17622.965,E2 -17622.965} C_VEL
LIN {X 0,Y 276.699,Z 392.016,A -85,B 0,C 180,E1 -17624.177,E2 -17624.177} C_VEL
LIN {X 0,Y 273.846,Z 392.372,A -85,B 0,C 180,E1 -17626.152,E2 -17626.152} C_VEL
LIN {X 0,Y 271.451,Z 392.666,A -85,B 0,C 180,E1 -17627.757,E2 -17627.757} C_VEL
LIN {X 0,Y 270.478,Z 392.786,A -85,B 0,C 180,E1 -17629.001,E2 -17629.001} C_VEL
LIN {X 0,Y 270.428,Z 392.793,A -85,B 0,C 180,E1 -17629.422,E2 -17629.422} C_VEL
LIN {X 0,Y 270.605,Z 392.776,A -85,B 0,C 180,E1 -17632.539,E2 -17632.539} C_VEL
LIN {X 0,Y 270.782,Z 392.754,A -85,B 0,C 180,E1 -17638.513,E2 -17638.513} C_VEL
LIN {X 0,Y 270.782,Z 392.746,A -85,B 0,C 180,E1 -17641.487,E2 -17641.487} C_VEL
LIN {X 0,Y 270.605,Z 392.77,A -85,B 0,C 180,E1 -17647.461,E2 -17647.461} C_VEL
LIN {X 0,Y 270.437,Z 392.795,A -85,B 0,C 180,E1 -17650.481,E2 -17650.481} C_VEL
LIN {X 0,Y 270.398,Z 392.799,A -85,B 0,C 180,E1 -17655.065,E2 -17655.065} C_VEL
LIN {X 0,Y 270.296,Z 392.807,A -85,B 0,C 180,E1 -17659.756,E2 -17659.756} C_VEL
LIN {X 0,Y 270.27,Z 392.815,A -85,B 0,C 180,E1 -17664.586,E2 -17664.586} C_VEL
LIN {X 0,Y 270.268,Z 392.817,A -85,B 0,C 180,E1 -17667.909,E2 -17667.909} C_VEL
LIN {X 0,Y 270.18,Z 392.828,A -85,B 0,C 180,E1 -17671.349,E2 -17671.349} C_VEL
LIN {X 0,Y 270.211,Z 392.825,A -85,B 0,C 180,E1 -17674.904,E2 -17674.904} C_VEL
LIN {X 0,Y 270.219,Z 392.824,A -85,B 0,C 180,E1 -17678.718,E2 -17678.718} C_VEL
LIN {X 0,Y 270.219,Z 392.823,A -85,B 0,C 180,E1 -17682.549,E2 -17682.549} C_VEL
LIN {X 0,Y 270.19,Z 392.828,A -85,B 0,C 180,E1 -17686.746,E2 -17686.746} C_VEL
LIN {X 0,Y 270.21,Z 392.826,A -85,B 0,C 180,E1 -17689.442,E2 -17689.442} C_VEL
LIN {X 0,Y 270.252,Z 392.933,A -85,B 0,C 180,E1 -17692.799,E2 -17692.799} C_VEL
LIN {X 0,Y 272.432,Z 402.16,A -85,B 0,C 180,E1 -17696.384,E2 -17696.384} C_VEL
LIN {X 0,Y 274.682,Z 412.349,A -85,B 0,C 180,E1 -17700.058,E2 -17700.058} C_VEL
LIN {X 0,Y 280.095,Z 425.728,A -85,B 0,C 180,E1 -17701.071,E2 -17701.071} C_VEL
LIN {X 0,Y 284.826,Z 455.076,A -85,B 0,C 180,E1 -17702.41,E2 -17702.41} C_VEL
LIN {X 0,Y 285.521,Z 462.119,A -85,B 0,C 180,E1 -17702.677,E2 -17702.677} C_VEL
LIN {X 0,Y 283.758,Z 521.004,A -85,B 0,C 180,E1 -17704.167,E2 -17704.167} C_VEL
LIN {X 0,Y 282.632,Z 534.92,A -85,B 0,C 180,E1 -17704.797,E2 -17704.797} C_VEL
LIN {X 0,Y 281.211,Z 547.37,A -85,B 0,C 180,E1 -17705.647,E2 -17705.647} C_VEL
LIN {X 0,Y 279.368,Z 560.064,A -85,B 0,C 180,E1 -17706.855,E2 -17706.855} C_VEL
LIN {X 0,Y 277.494,Z 571.354,A -85,B 0,C 180,E1 -17708.26,E2 -17708.26} C_VEL
LIN {X 0,Y 275.489,Z 581.525,A -85,B 0,C 180,E1 -17709.855,E2 -17709.855} C_VEL
LIN {X 0,Y 273.708,Z 590.862,A -85,B 0,C 180,E1 -17711.706,E2 -17711.706} C_VEL
LIN {X 0,Y 272.305,Z 598.281,A -85,B 0,C 180,E1 -17713.507,E2 -17713.507} C_VEL
LIN {X 0,Y 270.792,Z 605.725,A -85,B 0,C 180,E1 -17715.726,E2 -17715.726} C_VEL
LIN {X 0,Y 269.584,Z 611.706,A -85,B 0,C 180,E1 -17717.962,E2 -17717.962} C_VEL
LIN {X 0,Y 268.886,Z 616.442,A -85,B 0,C 180,E1 -17720.219,E2 -17720.219} C_VEL
LIN {X 0,Y 268.415,Z 620.062,A -85,B 0,C 180,E1 -17722.478,E2 -17722.478} C_VEL
LIN {X 0,Y 268.172,Z 622.724,A -85,B 0,C 180,E1 -17724.791,E2 -17724.791} C_VEL
LIN {X 0,Y 268.194,Z 624.338,A -85,B 0,C 180,E1 -17726.996,E2 -17726.996} C_VEL
LIN {X 0,Y 268.226,Z 624.951,A -85,B 0,C 180,E1 -17728.499,E2 -17728.499} C_VEL
LIN {X 0,Y 268.253,Z 625.166,A -85,B 0,C 180,E1 -17730,E2 -17730} C_VEL
LIN {X 0,Y 268.226,Z 624.942,A -85,B 0,C 180,E1 -17731.501,E2 -17731.501} C_VEL
LIN {X 0,Y 268.194,Z 624.325,A -85,B 0,C 180,E1 -17733.004,E2 -17733.004} C_VEL
LIN {X 0,Y 268.216,Z 622.6,A -85,B 0,C 180,E1 -17735.312,E2 -17735.312} C_VEL
LIN {X 0,Y 268.54,Z 618.945,A -85,B 0,C 180,E1 -17738.276,E2 -17738.276} C_VEL
LIN {X 0,Y 269.084,Z 614.946,A -85,B 0,C 180,E1 -17740.534,E2 -17740.534} C_VEL
LIN {X 0,Y 270.101,Z 608.803,A -85,B 0,C 180,E1 -17743.16,E2 -17743.16} C_VEL
LIN {X 0,Y 271.569,Z 602.109,A -85,B 0,C 180,E1 -17745.382,E2 -17745.382} C_VEL
LIN {X 0,Y 273.235,Z 593.803,A -85,B 0,C 180,E1 -17747.591,E2 -17747.591} C_VEL
LIN {X 0,Y 274.769,Z 585.284,A -85,B 0,C 180,E1 -17749.421,E2 -17749.421} C_VEL
LIN {X 0,Y 276.617,Z 575.952,A -85,B 0,C 180,E1 -17751.03,E2 -17751.03} C_VEL
LIN {X 0,Y 278.634,Z 564.377,A -85,B 0,C 180,E1 -17752.622,E2 -17752.622} C_VEL
LIN {X 0,Y 280.366,Z 552.975,A -85,B 0,C 180,E1 -17753.841,E2 -17753.841} C_VEL
LIN {X 0,Y 281.901,Z 541.249,A -85,B 0,C 180,E1 -17754.78,E2 -17754.78} C_VEL
LIN {X 0,Y 283.156,Z 528.644,A -85,B 0,C 180,E1 -17755.497,E2 -17755.497} C_VEL
LIN {X 0,Y 283.935,Z 515.785,A -85,B 0,C 180,E1 -17755.963,E2 -17755.963} C_VEL
LIN {X 0,Y 285.439,Z 460.533,A -85,B 0,C 180,E1 -17757.342,E2 -17757.342} C_VEL
LIN {X 0,Y 281.541,Z 434.027,A -85,B 0,C 180,E1 -17758.497,E2 -17758.497} C_VEL
LIN {X 0,Y 279.626,Z 424.426,A -85,B 0,C 180,E1 -17758.983,E2 -17758.983} C_VEL
LIN {X 0,Y 274.639,Z 412.126,A -85,B 0,C 180,E1 -17759.923,E2 -17759.923} C_VEL
LIN {X 0,Y 272.407,Z 402.049,A -85,B 0,C 180,E1 -17763.616,E2 -17763.616} C_VEL
LIN {X 0,Y 270.251,Z 392.817,A -85,B 0,C 180,E1 -17767.201,E2 -17767.201} C_VEL
LIN {X 0,Y 270.221,Z 392.825,A -85,B 0,C 180,E1 -17771.041,E2 -17771.041} C_VEL
LIN {X 0,Y 270.191,Z 392.815,A -85,B 0,C 180,E1 -17775.388,E2 -17775.388} C_VEL
LIN {X 0,Y 270.243,Z 392.82,A -85,B 0,C 180,E1 -17779.447,E2 -17779.447} C_VEL
LIN {X 0,Y 270.252,Z 392.821,A -85,B 0,C 180,E1 -17783.721,E2 -17783.721} C_VEL
LIN {X 0,Y 270.2,Z 392.822,A -85,B 0,C 180,E1 -17786.892,E2 -17786.892} C_VEL
LIN {X 0,Y 270.225,Z 392.82,A -85,B 0,C 180,E1 -17790.386,E2 -17790.386} C_VEL
LIN {X 0,Y 270.261,Z 392.818,A -85,B 0,C 180,E1 -17793.764,E2 -17793.764} C_VEL
LIN {X 0,Y 270.227,Z 392.816,A -85,B 0,C 180,E1 -17797.038,E2 -17797.038} C_VEL
LIN {X 0,Y 270.296,Z 392.813,A -85,B 0,C 180,E1 -17800.244,E2 -17800.244} C_VEL
LIN {X 0,Y 270.391,Z 392.801,A -85,B 0,C 180,E1 -17804.935,E2 -17804.935} C_VEL
LIN {X 0,Y 270.437,Z 392.787,A -85,B 0,C 180,E1 -17809.519,E2 -17809.519} C_VEL
LIN {X 0,Y 270.605,Z 392.775,A -85,B 0,C 180,E1 -17812.539,E2 -17812.539} C_VEL
LIN {X 0,Y 270.782,Z 392.747,A -85,B 0,C 180,E1 -17818.513,E2 -17818.513} C_VEL
LIN {X 0,Y 270.782,Z 392.753,A -85,B 0,C 180,E1 -17821.487,E2 -17821.487} C_VEL
LIN {X 0,Y 270.605,Z 392.776,A -85,B 0,C 180,E1 -17827.461,E2 -17827.461} C_VEL
LIN {X 0,Y 270.437,Z 392.796,A -85,B 0,C 180,E1 -17830.481,E2 -17830.481} C_VEL
LIN {X 0,Y 270.391,Z 392.804,A -85,B 0,C 180,E1 -17835.065,E2 -17835.065} C_VEL
LIN {X 0,Y 270.297,Z 392.804,A -85,B 0,C 180,E1 -17839.756,E2 -17839.756} C_VEL
LIN {X 0,Y 270.27,Z 392.815,A -85,B 0,C 180,E1 -17844.586,E2 -17844.586} C_VEL
LIN {X 0,Y 270.268,Z 392.816,A -85,B 0,C 180,E1 -17847.909,E2 -17847.909} C_VEL
LIN {X 0,Y 270.18,Z 392.822,A -85,B 0,C 180,E1 -17851.349,E2 -17851.349} C_VEL
LIN {X 0,Y 270.212,Z 392.825,A -85,B 0,C 180,E1 -17854.904,E2 -17854.904} C_VEL
LIN {X 0,Y 270.22,Z 392.826,A -85,B 0,C 180,E1 -17858.718,E2 -17858.718} C_VEL
LIN {X 0,Y 270.22,Z 392.827,A -85,B 0,C 180,E1 -17862.549,E2 -17862.549} C_VEL
LIN {X 0,Y 270.187,Z 392.829,A -85,B 0,C 180,E1 -17866.746,E2 -17866.746} C_VEL
LIN {X 0,Y 270.206,Z 392.826,A -85,B 0,C 180,E1 -17871.375,E2 -17871.375} C_VEL
LIN {X 0,Y 270.223,Z 392.826,A -85,B 0,C 180,E1 -17875.099,E2 -17875.099} C_VEL
LIN {X 0,Y 270.247,Z 393.007,A -85,B 0,C 180,E1 -17878.814,E2 -17878.814} C_VEL
LIN {X 0,Y 270.677,Z 394.97,A -85,B 0,C 180,E1 -17879.66,E2 -17879.66} C_VEL
LIN {X 0,Y 279.11,Z 412.753,A -85,B 0,C 180,E1 -17881.197,E2 -17881.197} C_VEL
LIN {X 0,Y 286.249,Z 430.788,A -85,B 0,C 180,E1 -17882.492,E2 -17882.492} C_VEL
LIN {X 0,Y 284.223,Z 501.091,A -85,B 0,C 180,E1 -17884.262,E2 -17884.262} C_VEL
LIN {X 0,Y 283.301,Z 514.437,A -85,B 0,C 180,E1 -17884.861,E2 -17884.861} C_VEL
LIN {X 0,Y 282.179,Z 527.173,A -85,B 0,C 180,E1 -17885.736,E2 -17885.736} C_VEL
LIN {X 0,Y 280.75,Z 538.483,A -85,B 0,C 180,E1 -17886.78,E2 -17886.78} C_VEL
LIN {X 0,Y 278.948,Z 550.113,A -85,B 0,C 180,E1 -17888.185,E2 -17888.185} C_VEL
LIN {X 0,Y 277.328,Z 560.345,A -85,B 0,C 180,E1 -17889.765,E2 -17889.765} C_VEL
LIN {X 0,Y 275.645,Z 569.072,A -85,B 0,C 180,E1 -17891.416,E2 -17891.416} C_VEL
LIN {X 0,Y 273.984,Z 576.927,A -85,B 0,C 180,E1 -17893.228,E2 -17893.228} C_VEL
LIN {X 0,Y 272.357,Z 584.598,A -85,B 0,C 180,E1 -17895.429,E2 -17895.429} C_VEL
LIN {X 0,Y 270.79,Z 591.639,A -85,B 0,C 180,E1 -17898.017,E2 -17898.017} C_VEL
LIN {X 0,Y 269.793,Z 596.325,A -85,B 0,C 180,E1 -17900.252,E2 -17900.252} C_VEL
LIN {X 0,Y 269.127,Z 599.907,A -85,B 0,C 180,E1 -17902.498,E2 -17902.498} C_VEL
LIN {X 0,Y 268.807,Z 601.757,A -85,B 0,C 180,E1 -17903.997,E2 -17903.997} C_VEL
LIN {X 0,Y 268.602,Z 603.146,A -85,B 0,C 180,E1 -17905.498,E2 -17905.498} C_VEL
LIN {X 0,Y 268.419,Z 604.136,A -85,B 0,C 180,E1 -17906.998,E2 -17906.998} C_VEL
LIN {X 0,Y 268.263,Z 604.975,A -85,B 0,C 180,E1 -17910,E2 -17910} C_VEL
LIN {X 0,Y 268.287,Z 604.783,A -85,B 0,C 180,E1 -17911.501,E2 -17911.501} C_VEL
LIN {X 0,Y 268.419,Z 604.198,A -85,B 0,C 180,E1 -17913.002,E2 -17913.002} C_VEL
LIN {X 0,Y 268.602,Z 603.232,A -85,B 0,C 180,E1 -17914.502,E2 -17914.502} C_VEL
LIN {X 0,Y 269.025,Z 600.813,A -85,B 0,C 180,E1 -17916.92,E2 -17916.92} C_VEL
LIN {X 0,Y 269.512,Z 597.828,A -85,B 0,C 180,E1 -17919.001,E2 -17919.001} C_VEL
LIN {X 0,Y 270.374,Z 593.584,A -85,B 0,C 180,E1 -17921.242,E2 -17921.242} C_VEL
LIN {X 0,Y 271.77,Z 587.155,A -85,B 0,C 180,E1 -17923.839,E2 -17923.839} C_VEL
LIN {X 0,Y 273.292,Z 580.085,A -85,B 0,C 180,E1 -17926.048,E2 -17926.048} C_VEL
LIN {X 0,Y 275.246,Z 571.271,A -85,B 0,C 180,E1 -17928.227,E2 -17928.227} C_VEL
LIN {X 0,Y 276.842,Z 563.136,A -85,B 0,C 180,E1 -17929.861,E2 -17929.861} C_VEL
LIN {X 0,Y 278.435,Z 553.426,A -85,B 0,C 180,E1 -17931.468,E2 -17931.468} C_VEL
LIN {X 0,Y 280.202,Z 542.628,A -85,B 0,C 180,E1 -17932.877,E2 -17932.877} C_VEL
LIN {X 0,Y 281.838,Z 530.507,A -85,B 0,C 180,E1 -17934.1,E2 -17934.1} C_VEL
LIN {X 0,Y 283.121,Z 517.797,A -85,B 0,C 180,E1 -17935.058,E2 -17935.058} C_VEL
LIN {X 0,Y 284.16,Z 505.084,A -85,B 0,C 180,E1 -17935.695,E2 -17935.695} C_VEL
LIN {X 0,Y 284.642,Z 488.85,A -85,B 0,C 180,E1 -17936.189,E2 -17936.189} C_VEL
LIN {X 0,Y 286.292,Z 430.895,A -85,B 0,C 180,E1 -17937.624,E2 -17937.624} C_VEL
LIN {X 0,Y 280.563,Z 416.158,A -85,B 0,C 180,E1 -17938.666,E2 -17938.666} C_VEL
LIN {X 0,Y 273.782,Z 401.38,A -85,B 0,C 180,E1 -17939.891,E2 -17939.891} C_VEL
LIN {X 0,Y 270.683,Z 394.978,A -85,B 0,C 180,E1 -17940.475,E2 -17940.475} C_VEL
LIN {X 0,Y 270.199,Z 392.826,A -85,B 0,C 180,E1 -17941.455,E2 -17941.455} C_VEL
LIN {X 0,Y 270.214,Z 392.826,A -85,B 0,C 180,E1 -17944.903,E2 -17944.903} C_VEL
LIN {X 0,Y 270.221,Z 392.824,A -85,B 0,C 180,E1 -17948.716,E2 -17948.716} C_VEL
LIN {X 0,Y 270.187,Z 392.826,A -85,B 0,C 180,E1 -17953.254,E2 -17953.254} C_VEL
LIN {X 0,Y 270.22,Z 392.811,A -85,B 0,C 180,E1 -17957.451,E2 -17957.451} C_VEL
LIN {X 0,Y 270.242,Z 392.824,A -85,B 0,C 180,E1 -17961.38,E2 -17961.38} C_VEL
LIN {X 0,Y 270.212,Z 392.826,A -85,B 0,C 180,E1 -17965.096,E2 -17965.096} C_VEL
LIN {X 0,Y 270.197,Z 392.828,A -85,B 0,C 180,E1 -17969.13,E2 -17969.13} C_VEL
LIN {X 0,Y 270.261,Z 392.817,A -85,B 0,C 180,E1 -17972.145,E2 -17972.145} C_VEL
LIN {X 0,Y 270.273,Z 392.816,A -85,B 0,C 180,E1 -17975.519,E2 -17975.519} C_VEL
LIN {X 0,Y 270.297,Z 392.814,A -85,B 0,C 180,E1 -17980.244,E2 -17980.244} C_VEL
LIN {X 0,Y 270.391,Z 392.802,A -85,B 0,C 180,E1 -17984.935,E2 -17984.935} C_VEL
LIN {X 0,Y 270.428,Z 392.793,A -85,B 0,C 180,E1 -17989.422,E2 -17989.422} C_VEL
LIN {X 0,Y 270.161,Z 392.831,A -85,B 0,C 180,E1 -17990.255,E2 -17990.255} C_VEL
LIN {X 0,Y 268.823,Z 393.001,A -85,B 0,C 180,E1 -17991.483,E2 -17991.483} C_VEL
LIN {X 0,Y 264.458,Z 393.538,A -85,B 0,C 180,E1 -17994.343,E2 -17994.343} C_VEL
LIN {X 0,Y 263.471,Z 393.658,A -85,B 0,C 180,E1 -17995.623,E2 -17995.623} C_VEL
LIN {X 0,Y 263.43,Z 393.661,A -85,B 0,C 180,E1 -17996.056,E2 -17996.056} C_VEL
LIN {X 0,Y 263.746,Z 393.63,A -85,B 0,C 180,E1 -17998.473,E2 -17998.473} C_VEL
LIN {X 0,Y 263.747,Z 393.621,A -85,B 0,C 180,E1 -18001.527,E2 -18001.527} C_VEL
LIN {X 0,Y 263.566,Z 393.645,A -85,B 0,C 180,E1 -18007.662,E2 -18007.662} C_VEL
LIN {X 0,Y 263.369,Z 393.677,A -85,B 0,C 180,E1 -18010.766,E2 -18010.766} C_VEL
LIN {X 0,Y 263.346,Z 393.679,A -85,B 0,C 180,E1 -18015.478,E2 -18015.478} C_VEL
LIN {X 0,Y 263.259,Z 393.685,A -85,B 0,C 180,E1 -18020.307,E2 -18020.307} C_VEL
LIN {X 0,Y 263.205,Z 393.696,A -85,B 0,C 180,E1 -18025.292,E2 -18025.292} C_VEL
LIN {X 0,Y 263.176,Z 393.703,A -85,B 0,C 180,E1 -18028.73,E2 -18028.73} C_VEL
LIN {X 0,Y 263.129,Z 393.707,A -85,B 0,C 180,E1 -18032.289,E2 -18032.289} C_VEL
LIN {X 0,Y 263.185,Z 393.698,A -85,B 0,C 180,E1 -18035.979,E2 -18035.979} C_VEL
LIN {X 0,Y 263.157,Z 393.701,A -85,B 0,C 180,E1 -18039.863,E2 -18039.863} C_VEL
LIN {X 0,Y 263.142,Z 393.702,A -85,B 0,C 180,E1 -18043.98,E2 -18043.98} C_VEL
LIN {X 0,Y 263.153,Z 393.704,A -85,B 0,C 180,E1 -18048.4,E2 -18048.4} C_VEL
LIN {X 0,Y 263.196,Z 393.76,A -85,B 0,C 180,E1 -18052.051,E2 -18052.051} C_VEL
LIN {X 0,Y 265.292,Z 402.484,A -85,B 0,C 180,E1 -18055.58,E2 -18055.58} C_VEL
LIN {X 0,Y 267.342,Z 411.832,A -85,B 0,C 180,E1 -18059.139,E2 -18059.139} C_VEL
LIN {X 0,Y 273.976,Z 427.843,A -85,B 0,C 180,E1 -18060.431,E2 -18060.431} C_VEL
LIN {X 0,Y 277.558,Z 449.207,A -85,B 0,C 180,E1 -18061.462,E2 -18061.462} C_VEL
LIN {X 0,Y 279.228,Z 461.873,A -85,B 0,C 180,E1 -18062.008,E2 -18062.008} C_VEL
LIN {X 0,Y 277.388,Z 520.751,A -85,B 0,C 180,E1 -18063.529,E2 -18063.529} C_VEL
LIN {X 0,Y 276.227,Z 534.662,A -85,B 0,C 180,E1 -18064.17,E2 -18064.17} C_VEL
LIN {X 0,Y 274.765,Z 547.11,A -85,B 0,C 180,E1 -18065.037,E2 -18065.037} C_VEL
LIN {X 0,Y 272.858,Z 559.802,A -85,B 0,C 180,E1 -18066.269,E2 -18066.269} C_VEL
LIN {X 0,Y 270.878,Z 571.089,A -85,B 0,C 180,E1 -18067.701,E2 -18067.701} C_VEL
LIN {X 0,Y 268.83,Z 581.261,A -85,B 0,C 180,E1 -18069.334,E2 -18069.334} C_VEL
LIN {X 0,Y 266.952,Z 590.43,A -85,B 0,C 180,E1 -18071.186,E2 -18071.186} C_VEL
LIN {X 0,Y 265.495,Z 598.016,A -85,B 0,C 180,E1 -18073.072,E2 -18073.072} C_VEL
LIN {X 0,Y 263.888,Z 605.458,A -85,B 0,C 180,E1 -18075.345,E2 -18075.345} C_VEL
LIN {X 0,Y 262.599,Z 611.438,A -85,B 0,C 180,E1 -18077.637,E2 -18077.637} C_VEL
LIN {X 0,Y 261.842,Z 616.174,A -85,B 0,C 180,E1 -18079.953,E2 -18079.953} C_VEL
LIN {X 0,Y 261.349,Z 619.795,A -85,B 0,C 180,E1 -18082.273,E2 -18082.273} C_VEL
LIN {X 0,Y 261.085,Z 622.66,A -85,B 0,C 180,E1 -18084.863,E2 -18084.863} C_VEL
LIN {X 0,Y 261.106,Z 624.071,A -85,B 0,C 180,E1 -18086.914,E2 -18086.914} C_VEL
LIN {X 0,Y 261.151,Z 624.685,A -85,B 0,C 180,E1 -18088.458,E2 -18088.458} C_VEL
LIN {X 0,Y 261.177,Z 624.899,A -85,B 0,C 180,E1 -18090,E2 -18090} C_VEL
LIN {X 0,Y 261.151,Z 624.676,A -85,B 0,C 180,E1 -18091.542,E2 -18091.542} C_VEL
LIN {X 0,Y 261.106,Z 624.057,A -85,B 0,C 180,E1 -18093.086,E2 -18093.086} C_VEL
LIN {X 0,Y 261.132,Z 622.528,A -85,B 0,C 180,E1 -18095.249,E2 -18095.249} C_VEL
LIN {X 0,Y 261.336,Z 619.754,A -85,B 0,C 180,E1 -18097.727,E2 -18097.727} C_VEL
LIN {X 0,Y 261.84,Z 616.115,A -85,B 0,C 180,E1 -18100.047,E2 -18100.047} C_VEL
LIN {X 0,Y 262.594,Z 611.364,A -85,B 0,C 180,E1 -18102.363,E2 -18102.363} C_VEL
LIN {X 0,Y 264.158,Z 604.246,A -85,B 0,C 180,E1 -18105.034,E2 -18105.034} C_VEL
LIN {X 0,Y 265.807,Z 596.655,A -85,B 0,C 180,E1 -18107.268,E2 -18107.268} C_VEL
LIN {X 0,Y 267.375,Z 588.614,A -85,B 0,C 180,E1 -18109.18,E2 -18109.18} C_VEL
LIN {X 0,Y 269.269,Z 578.97,A -85,B 0,C 180,E1 -18111.031,E2 -18111.031} C_VEL
LIN {X 0,Y 271.347,Z 568.284,A -85,B 0,C 180,E1 -18112.66,E2 -18112.66} C_VEL
LIN {X 0,Y 273.132,Z 557.953,A -85,B 0,C 180,E1 -18113.907,E2 -18113.907} C_VEL
LIN {X 0,Y 274.758,Z 546.736,A -85,B 0,C 180,E1 -18114.964,E2 -18114.964} C_VEL
LIN {X 0,Y 276.209,Z 534.132,A -85,B 0,C 180,E1 -18115.832,E2 -18115.832} C_VEL
LIN {X 0,Y 277.284,Z 521.11,A -85,B 0,C 180,E1 -18116.431,E2 -18116.431} C_VEL
LIN {X 0,Y 279.089,Z 460.865,A -85,B 0,C 180,E1 -18118.001,E2 -18118.001} C_VEL
LIN {X 0,Y 274.881,Z 432.556,A -85,B 0,C 180,E1 -18119.288,E2 -18119.288} C_VEL
LIN {X 0,Y 273.417,Z 426.303,A -85,B 0,C 180,E1 -18119.642,E2 -18119.642} C_VEL
LIN {X 0,Y 267.342,Z 411.785,A -85,B 0,C 180,E1 -18120.838,E2 -18120.838} C_VEL
LIN {X 0,Y 265.093,Z 401.581,A -85,B 0,C 180,E1 -18124.729,E2 -18124.729} C_VEL
LIN {X 0,Y 263.184,Z 393.697,A -85,B 0,C 180,E1 -18128.011,E2 -18128.011} C_VEL
LIN {X 0,Y 263.147,Z 393.704,A -85,B 0,C 180,E1 -18131.888,E2 -18131.888} C_VEL
LIN {X 0,Y 263.144,Z 393.696,A -85,B 0,C 180,E1 -18136.145,E2 -18136.145} C_VEL
LIN {X 0,Y 263.157,Z 393.704,A -85,B 0,C 180,E1 -18140.137,E2 -18140.137} C_VEL
LIN {X 0,Y 263.185,Z 393.701,A -85,B 0,C 180,E1 -18144.022,E2 -18144.022} C_VEL
LIN {X 0,Y 263.129,Z 393.706,A -85,B 0,C 180,E1 -18147.711,E2 -18147.711} C_VEL
LIN {X 0,Y 263.197,Z 393.693,A -85,B 0,C 180,E1 -18151.782,E2 -18151.782} C_VEL
LIN {X 0,Y 263.222,Z 393.693,A -85,B 0,C 180,E1 -18155.2,E2 -18155.2} C_VEL
LIN {X 0,Y 263.259,Z 393.691,A -85,B 0,C 180,E1 -18159.693,E2 -18159.693} C_VEL
LIN {X 0,Y 263.339,Z 393.677,A -85,B 0,C 180,E1 -18164.521,E2 -18164.521} C_VEL
LIN {X 0,Y 263.369,Z 393.668,A -85,B 0,C 180,E1 -18169.234,E2 -18169.234} C_VEL
LIN {X 0,Y 263.566,Z 393.651,A -85,B 0,C 180,E1 -18172.338,E2 -18172.338} C_VEL
LIN {X 0,Y 263.746,Z 393.623,A -85,B 0,C 180,E1 -18178.473,E2 -18178.473} C_VEL
LIN {X 0,Y 263.747,Z 393.63,A -85,B 0,C 180,E1 -18181.527,E2 -18181.527} C_VEL
LIN {X 0,Y 263.567,Z 393.652,A -85,B 0,C 180,E1 -18187.662,E2 -18187.662} C_VEL
LIN {X 0,Y 263.369,Z 393.672,A -85,B 0,C 180,E1 -18190.766,E2 -18190.766} C_VEL
LIN {X 0,Y 263.34,Z 393.681,A -85,B 0,C 180,E1 -18195.479,E2 -18195.479} C_VEL
LIN {X 0,Y 263.259,Z 393.683,A -85,B 0,C 180,E1 -18200.307,E2 -18200.307} C_VEL
LIN {X 0,Y 263.204,Z 393.69,A -85,B 0,C 180,E1 -18205.292,E2 -18205.292} C_VEL
LIN {X 0,Y 263.176,Z 393.704,A -85,B 0,C 180,E1 -18208.73,E2 -18208.73} C_VEL
LIN {X 0,Y 263.13,Z 393.701,A -85,B 0,C 180,E1 -18212.289,E2 -18212.289} C_VEL
LIN {X 0,Y 263.187,Z 393.699,A -85,B 0,C 180,E1 -18215.978,E2 -18215.978} C_VEL
LIN {X 0,Y 263.158,Z 393.705,A -85,B 0,C 180,E1 -18219.863,E2 -18219.863} C_VEL
LIN {X 0,Y 263.143,Z 393.706,A -85,B 0,C 180,E1 -18223.98,E2 -18223.98} C_VEL
LIN {X 0,Y 263.128,Z 393.707,A -85,B 0,C 180,E1 -18228.406,E2 -18228.406} C_VEL
LIN {X 0,Y 263.165,Z 393.706,A -85,B 0,C 180,E1 -18232.105,E2 -18232.105} C_VEL
LIN {X 0,Y 263.183,Z 393.703,A -85,B 0,C 180,E1 -18235.891,E2 -18235.891} C_VEL
LIN {X 0,Y 263.156,Z 393.781,A -85,B 0,C 180,E1 -18238.07,E2 -18238.07} C_VEL
LIN {X 0,Y 263.594,Z 395.448,A -85,B 0,C 180,E1 -18238.763,E2 -18238.763} C_VEL
LIN {X 0,Y 272.954,Z 414.935,A -85,B 0,C 180,E1 -18240.541,E2 -18240.541} C_VEL
LIN {X 0,Y 279.919,Z 432.401,A -85,B 0,C 180,E1 -18241.852,E2 -18241.852} C_VEL
LIN {X 0,Y 278.327,Z 488.254,A -85,B 0,C 180,E1 -18243.271,E2 -18243.271} C_VEL
LIN {X 0,Y 277.654,Z 504.798,A -85,B 0,C 180,E1 -18243.758,E2 -18243.758} C_VEL
LIN {X 0,Y 276.664,Z 517.725,A -85,B 0,C 180,E1 -18244.416,E2 -18244.416} C_VEL
LIN {X 0,Y 275.453,Z 529.534,A -85,B 0,C 180,E1 -18245.305,E2 -18245.305} C_VEL
LIN {X 0,Y 273.754,Z 541.915,A -85,B 0,C 180,E1 -18246.552,E2 -18246.552} C_VEL
LIN {X 0,Y 271.932,Z 552.948,A -85,B 0,C 180,E1 -18247.992,E2 -18247.992} C_VEL
LIN {X 0,Y 270.428,Z 562.202,A -85,B 0,C 180,E1 -18249.528,E2 -18249.528} C_VEL
LIN {X 0,Y 268.562,Z 571.03,A -85,B 0,C 180,E1 -18251.303,E2 -18251.303} C_VEL
LIN {X 0,Y 266.575,Z 579.927,A -85,B 0,C 180,E1 -18253.536,E2 -18253.536} C_VEL
LIN {X 0,Y 264.948,Z 587.084,A -85,B 0,C 180,E1 -18255.797,E2 -18255.797} C_VEL
LIN {X 0,Y 263.854,Z 591.907,A -85,B 0,C 180,E1 -18257.697,E2 -18257.697} C_VEL
LIN {X 0,Y 262.8,Z 596.593,A -85,B 0,C 180,E1 -18259.99,E2 -18259.99} C_VEL
LIN {X 0,Y 262.08,Z 600.175,A -85,B 0,C 180,E1 -18262.295,E2 -18262.295} C_VEL
LIN {X 0,Y 261.743,Z 602.025,A -85,B 0,C 180,E1 -18263.835,E2 -18263.835} C_VEL
LIN {X 0,Y 261.532,Z 603.414,A -85,B 0,C 180,E1 -18265.376,E2 -18265.376} C_VEL
LIN {X 0,Y 261.357,Z 604.403,A -85,B 0,C 180,E1 -18266.917,E2 -18266.917} C_VEL
LIN {X 0,Y 261.187,Z 605.242,A -85,B 0,C 180,E1 -18270,E2 -18270} C_VEL
LIN {X 0,Y 261.215,Z 605.049,A -85,B 0,C 180,E1 -18271.542,E2 -18271.542} C_VEL
LIN {X 0,Y 261.356,Z 604.463,A -85,B 0,C 180,E1 -18273.083,E2 -18273.083} C_VEL
LIN {X 0,Y 261.532,Z 603.498,A -85,B 0,C 180,E1 -18274.624,E2 -18274.624} C_VEL
LIN {X 0,Y 261.953,Z 601.278,A -85,B 0,C 180,E1 -18276.933,E2 -18276.933} C_VEL
LIN {X 0,Y 262.514,Z 598.094,A -85,B 0,C 180,E1 -18279.243,E2 -18279.243} C_VEL
LIN {X 0,Y 263.413,Z 593.85,A -85,B 0,C 180,E1 -18281.543,E2 -18281.543} C_VEL
LIN {X 0,Y 264.895,Z 587.42,A -85,B 0,C 180,E1 -18284.206,E2 -18284.206} C_VEL
LIN {X 0,Y 266.462,Z 580.351,A -85,B 0,C 180,E1 -18286.471,E2 -18286.471} C_VEL
LIN {X 0,Y 268.518,Z 571.535,A -85,B 0,C 180,E1 -18288.7,E2 -18288.7} C_VEL
LIN {X 0,Y 270.364,Z 562.013,A -85,B 0,C 180,E1 -18290.641,E2 -18290.641} C_VEL
LIN {X 0,Y 272.262,Z 551.184,A -85,B 0,C 180,E1 -18292.379,E2 -18292.379} C_VEL
LIN {X 0,Y 274.181,Z 539.736,A -85,B 0,C 180,E1 -18293.81,E2 -18293.81} C_VEL
LIN {X 0,Y 275.799,Z 527.722,A -85,B 0,C 180,E1 -18294.964,E2 -18294.964} C_VEL
LIN {X 0,Y 277.041,Z 514.321,A -85,B 0,C 180,E1 -18295.9,E2 -18295.9} C_VEL
LIN {X 0,Y 277.947,Z 501.919,A -85,B 0,C 180,E1 -18296.465,E2 -18296.465} C_VEL
LIN {X 0,Y 279.34,Z 458.042,A -85,B 0,C 180,E1 -18297.605,E2 -18297.605} C_VEL
LIN {X 0,Y 280.029,Z 432.667,A -85,B 0,C 180,E1 -18298.253,E2 -18298.253} C_VEL
LIN {X 0,Y 273.52,Z 416.216,A -85,B 0,C 180,E1 -18299.482,E2 -18299.482} C_VEL
LIN {X 0,Y 266.568,Z 401.549,A -85,B 0,C 180,E1 -18300.79,E2 -18300.79} C_VEL
LIN {X 0,Y 263.521,Z 395.23,A -85,B 0,C 180,E1 -18301.413,E2 -18301.413} C_VEL
LIN {X 0,Y 263.155,Z 393.71,A -85,B 0,C 180,E1 -18302.145,E2 -18302.145} C_VEL
LIN {X 0,Y 263.187,Z 393.702,A -85,B 0,C 180,E1 -18305.977,E2 -18305.977} C_VEL
LIN {X 0,Y 263.116,Z 393.71,A -85,B 0,C 180,E1 -18309.869,E2 -18309.869} C_VEL
LIN {X 0,Y 263.137,Z 393.709,A -85,B 0,C 180,E1 -18313.98,E2 -18313.98} C_VEL
LIN {X 0,Y 263.171,Z 393.694,A -85,B 0,C 180,E1 -18318.394,E2 -18318.394} C_VEL
LIN {X 0,Y 263.186,Z 393.696,A -85,B 0,C 180,E1 -18322.107,E2 -18322.107} C_VEL
LIN {X 0,Y 263.181,Z 393.698,A -85,B 0,C 180,E1 -18325.89,E2 -18325.89} C_VEL
LIN {X 0,Y 263.147,Z 393.707,A -85,B 0,C 180,E1 -18329.506,E2 -18329.506} C_VEL
LIN {X 0,Y 263.189,Z 393.698,A -85,B 0,C 180,E1 -18333.002,E2 -18333.002} C_VEL
LIN {X 0,Y 263.179,Z 393.695,A -85,B 0,C 180,E1 -18336.386,E2 -18336.386} C_VEL
LIN {X 0,Y 263.259,Z 393.693,A -85,B 0,C 180,E1 -18339.693,E2 -18339.693} C_VEL
LIN {X 0,Y 263.34,Z 393.679,A -85,B 0,C 180,E1 -18344.521,E2 -18344.521} C_VEL
LIN {X 0,Y 263.382,Z 393.669,A -85,B 0,C 180,E1 -18349.445,E2 -18349.445} C_VEL
LIN {X 0,Y 263.567,Z 393.652,A -85,B 0,C 180,E1 -18352.338,E2 -18352.338} C_VEL
LIN {X 0,Y 263.43,Z 393.661,A -85,B 0,C 180,E1 -18356.056,E2 -18356.056} C_VEL
LIN {X 0,Y 262.892,Z 393.737,A -85,B 0,C 180,E1 -18357.335,E2 -18357.335} C_VEL
LIN {X 0,Y 260.164,Z 394.077,A -85,B 0,C 180,E1 -18359.423,E2 -18359.423} C_VEL
LIN {X 0,Y 256.895,Z 394.473,A -85,B 0,C 180,E1 -18361.992,E2 -18361.992} C_VEL
LIN {X 0,Y 256.517,Z 394.523,A -85,B 0,C 180,E1 -18362.881,E2 -18362.881} C_VEL
LIN {X 0,Y 256.534,Z 394.52,A -85,B 0,C 180,E1 -18367.873,E2 -18367.873} C_VEL
LIN {X 0,Y 256.305,Z 394.56,A -85,B 0,C 180,E1 -18371.066,E2 -18371.066} C_VEL
LIN {X 0,Y 256.295,Z 394.556,A -85,B 0,C 180,E1 -18375.915,E2 -18375.915} C_VEL
LIN {X 0,Y 256.162,Z 394.573,A -85,B 0,C 180,E1 -18380.896,E2 -18380.896} C_VEL
LIN {X 0,Y 256.184,Z 394.57,A -85,B 0,C 180,E1 -18385.139,E2 -18385.139} C_VEL
LIN {X 0,Y 256.11,Z 394.58,A -85,B 0,C 180,E1 -18389.6,E2 -18389.6} C_VEL
LIN {X 0,Y 256.081,Z 394.578,A -85,B 0,C 180,E1 -18393.291,E2 -18393.291} C_VEL
LIN {X 0,Y 256.136,Z 394.572,A -85,B 0,C 180,E1 -18397.279,E2 -18397.279} C_VEL
LIN {X 0,Y 256.101,Z 394.581,A -85,B 0,C 180,E1 -18401.194,E2 -18401.194} C_VEL
LIN {X 0,Y 256.071,Z 394.586,A -85,B 0,C 180,E1 -18405.527,E2 -18405.527} C_VEL
LIN {X 0,Y 256.083,Z 394.584,A -85,B 0,C 180,E1 -18408.803,E2 -18408.803} C_VEL
LIN {X 0,Y 256.15,Z 394.785,A -85,B 0,C 180,E1 -18411.335,E2 -18411.335} C_VEL
LIN {X 0,Y 258.156,Z 402.903,A -85,B 0,C 180,E1 -18414.757,E2 -18414.757} C_VEL
LIN {X 0,Y 260.14,Z 411.783,A -85,B 0,C 180,E1 -18418.196,E2 -18418.196} C_VEL
LIN {X 0,Y 267.936,Z 429.983,A -85,B 0,C 180,E1 -18419.768,E2 -18419.768} C_VEL
LIN {X 0,Y 270.862,Z 447.246,A -85,B 0,C 180,E1 -18420.639,E2 -18420.639} C_VEL
LIN {X 0,Y 272.947,Z 462.588,A -85,B 0,C 180,E1 -18421.333,E2 -18421.333} C_VEL
LIN {X 0,Y 271.062,Z 520.498,A -85,B 0,C 180,E1 -18422.861,E2 -18422.861} C_VEL
LIN {X 0,Y 269.864,Z 534.404,A -85,B 0,C 180,E1 -18423.515,E2 -18423.515} C_VEL
LIN {X 0,Y 268.343,Z 546.849,A -85,B 0,C 180,E1 -18424.397,E2 -18424.397} C_VEL
LIN {X 0,Y 266.368,Z 559.539,A -85,B 0,C 180,E1 -18425.654,E2 -18425.654} C_VEL
LIN {X 0,Y 264.285,Z 570.824,A -85,B 0,C 180,E1 -18427.114,E2 -18427.114} C_VEL
LIN {X 0,Y 262.174,Z 580.995,A -85,B 0,C 180,E1 -18428.784,E2 -18428.784} C_VEL
LIN {X 0,Y 260.204,Z 590.164,A -85,B 0,C 180,E1 -18430.679,E2 -18430.679} C_VEL
LIN {X 0,Y 258.702,Z 597.75,A -85,B 0,C 180,E1 -18432.613,E2 -18432.613} C_VEL
LIN {X 0,Y 257.006,Z 605.192,A -85,B 0,C 180,E1 -18434.943,E2 -18434.943} C_VEL
LIN {X 0,Y 255.62,Z 611.171,A -85,B 0,C 180,E1 -18437.294,E2 -18437.294} C_VEL
LIN {X 0,Y 254.808,Z 615.906,A -85,B 0,C 180,E1 -18439.672,E2 -18439.672} C_VEL
LIN {X 0,Y 254.307,Z 619.528,A -85,B 0,C 180,E1 -18442.058,E2 -18442.058} C_VEL
LIN {X 0,Y 253.99,Z 622.599,A -85,B 0,C 180,E1 -18444.961,E2 -18444.961} C_VEL
LIN {X 0,Y 254.001,Z 623.804,A -85,B 0,C 180,E1 -18446.828,E2 -18446.828} C_VEL
LIN {X 0,Y 254.077,Z 624.418,A -85,B 0,C 180,E1 -18448.415,E2 -18448.415} C_VEL
LIN {X 0,Y 254.102,Z 624.633,A -85,B 0,C 180,E1 -18450,E2 -18450} C_VEL
LIN {X 0,Y 254.077,Z 624.409,A -85,B 0,C 180,E1 -18451.585,E2 -18451.585} C_VEL
LIN {X 0,Y 254.002,Z 623.789,A -85,B 0,C 180,E1 -18453.172,E2 -18453.172} C_VEL
LIN {X 0,Y 254.022,Z 622.513,A -85,B 0,C 180,E1 -18455.119,E2 -18455.119} C_VEL
LIN {X 0,Y 254.298,Z 619.486,A -85,B 0,C 180,E1 -18457.943,E2 -18457.943} C_VEL
LIN {X 0,Y 254.806,Z 615.846,A -85,B 0,C 180,E1 -18460.328,E2 -18460.328} C_VEL
LIN {X 0,Y 255.616,Z 611.094,A -85,B 0,C 180,E1 -18462.706,E2 -18462.706} C_VEL
LIN {X 0,Y 257.284,Z 603.976,A -85,B 0,C 180,E1 -18465.446,E2 -18465.446} C_VEL
LIN {X 0,Y 258.981,Z 596.554,A -85,B 0,C 180,E1 -18467.69,E2 -18467.69} C_VEL
LIN {X 0,Y 260.63,Z 588.339,A -85,B 0,C 180,E1 -18469.698,E2 -18469.698} C_VEL
LIN {X 0,Y 262.643,Z 578.699,A -85,B 0,C 180,E1 -18471.588,E2 -18471.588} C_VEL
LIN {X 0,Y 264.806,Z 568.012,A -85,B 0,C 180,E1 -18473.252,E2 -18473.252} C_VEL
LIN {X 0,Y 266.659,Z 557.681,A -85,B 0,C 180,E1 -18474.525,E2 -18474.525} C_VEL
LIN {X 0,Y 268.338,Z 546.462,A -85,B 0,C 180,E1 -18475.603,E2 -18475.603} C_VEL
LIN {X 0,Y 269.848,Z 533.857,A -85,B 0,C 180,E1 -18476.487,E2 -18476.487} C_VEL
LIN {X 0,Y 270.951,Z 520.829,A -85,B 0,C 180,E1 -18477.099,E2 -18477.099} C_VEL
LIN {X 0,Y 272.823,Z 461.945,A -85,B 0,C 180,E1 -18478.663,E2 -18478.663} C_VEL
LIN {X 0,Y 268.937,Z 435.206,A -85,B 0,C 180,E1 -18479.912,E2 -18479.912} C_VEL
LIN {X 0,Y 267.741,Z 429.572,A -85,B 0,C 180,E1 -18480.229,E2 -18480.229} C_VEL
LIN {X 0,Y 261.476,Z 414.917,A -85,B 0,C 180,E1 -18481.482,E2 -18481.482} C_VEL
LIN {X 0,Y 260.009,Z 411.387,A -85,B 0,C 180,E1 -18481.838,E2 -18481.838} C_VEL
LIN {X 0,Y 257.786,Z 401.114,A -85,B 0,C 180,E1 -18485.922,E2 -18485.922} C_VEL
LIN {X 0,Y 256.129,Z 394.581,A -85,B 0,C 180,E1 -18488.782,E2 -18488.782} C_VEL
LIN {X 0,Y 256.093,Z 394.582,A -85,B 0,C 180,E1 -18493.319,E2 -18493.319} C_VEL
LIN {X 0,Y 256.122,Z 394.581,A -85,B 0,C 180,E1 -18497.805,E2 -18497.805} C_VEL
LIN {X 0,Y 256.106,Z 394.582,A -85,B 0,C 180,E1 -18500.864,E2 -18500.864} C_VEL
LIN {X 0,Y 256.117,Z 394.581,A -85,B 0,C 180,E1 -18504.813,E2 -18504.813} C_VEL
LIN {X 0,Y 256.088,Z 394.583,A -85,B 0,C 180,E1 -18508.572,E2 -18508.572} C_VEL
LIN {X 0,Y 256.138,Z 394.573,A -85,B 0,C 180,E1 -18512.196,E2 -18512.196} C_VEL
LIN {X 0,Y 256.162,Z 394.568,A -85,B 0,C 180,E1 -18515.699,E2 -18515.699} C_VEL
LIN {X 0,Y 256.162,Z 394.575,A -85,B 0,C 180,E1 -18519.104,E2 -18519.104} C_VEL
LIN {X 0,Y 256.289,Z 394.554,A -85,B 0,C 180,E1 -18524.084,E2 -18524.084} C_VEL
LIN {X 0,Y 256.305,Z 394.549,A -85,B 0,C 180,E1 -18528.934,E2 -18528.934} C_VEL
LIN {X 0,Y 256.534,Z 394.527,A -85,B 0,C 180,E1 -18532.127,E2 -18532.127} C_VEL
LIN {X 0,Y 256.709,Z 394.499,A -85,B 0,C 180,E1 -18538.431,E2 -18538.431} C_VEL
LIN {X 0,Y 256.71,Z 394.506,A -85,B 0,C 180,E1 -18541.569,E2 -18541.569} C_VEL
LIN {X 0,Y 256.534,Z 394.528,A -85,B 0,C 180,E1 -18547.873,E2 -18547.873} C_VEL
LIN {X 0,Y 256.305,Z 394.549,A -85,B 0,C 180,E1 -18551.066,E2 -18551.066} C_VEL
LIN {X 0,Y 256.29,Z 394.559,A -85,B 0,C 180,E1 -18555.916,E2 -18555.916} C_VEL
LIN {X 0,Y 256.162,Z 394.571,A -85,B 0,C 180,E1 -18560.896,E2 -18560.896} C_VEL
LIN {X 0,Y 256.184,Z 394.565,A -85,B 0,C 180,E1 -18565.139,E2 -18565.139} C_VEL
LIN {X 0,Y 256.11,Z 394.581,A -85,B 0,C 180,E1 -18569.6,E2 -18569.6} C_VEL
LIN {X 0,Y 256.082,Z 394.584,A -85,B 0,C 180,E1 -18573.291,E2 -18573.291} C_VEL
LIN {X 0,Y 256.138,Z 394.575,A -85,B 0,C 180,E1 -18577.279,E2 -18577.279} C_VEL
LIN {X 0,Y 256.101,Z 394.578,A -85,B 0,C 180,E1 -18581.195,E2 -18581.195} C_VEL
LIN {X 0,Y 256.071,Z 394.584,A -85,B 0,C 180,E1 -18585.528,E2 -18585.528} C_VEL
LIN {X 0,Y 256.06,Z 394.589,A -85,B 0,C 180,E1 -18588.799,E2 -18588.799} C_VEL
LIN {X 0,Y 256.144,Z 394.579,A -85,B 0,C 180,E1 -18592.871,E2 -18592.871} C_VEL
LIN {X 0,Y 256.108,Z 394.685,A -85,B 0,C 180,E1 -18597.344,E2 -18597.344} C_VEL
LIN {X 0,Y 256.372,Z 395.803,A -85,B 0,C 180,E1 -18597.779,E2 -18597.779} C_VEL
LIN {X 0,Y 265.803,Z 414.771,A -85,B 0,C 180,E1 -18599.651,E2 -18599.651} C_VEL
LIN {X 0,Y 272.465,Z 430.965,A -85,B 0,C 180,E1 -18600.958,E2 -18600.958} C_VEL
LIN {X 0,Y 273.765,Z 434.852,A -85,B 0,C 180,E1 -18601.225,E2 -18601.225} C_VEL
LIN {X 0,Y 271.534,Z 501.657,A -85,B 0,C 180,E1 -18602.964,E2 -18602.964} C_VEL
LIN {X 0,Y 270.564,Z 514.99,A -85,B 0,C 180,E1 -18603.588,E2 -18603.588} C_VEL
LIN {X 0,Y 269.318,Z 527.721,A -85,B 0,C 180,E1 -18604.496,E2 -18604.496} C_VEL
LIN {X 0,Y 267.802,Z 539.027,A -85,B 0,C 180,E1 -18605.586,E2 -18605.586} C_VEL
LIN {X 0,Y 265.861,Z 550.654,A -85,B 0,C 180,E1 -18607.051,E2 -18607.051} C_VEL
LIN {X 0,Y 264.04,Z 560.826,A -85,B 0,C 180,E1 -18608.687,E2 -18608.687} C_VEL
LIN {X 0,Y 262.248,Z 569.611,A -85,B 0,C 180,E1 -18610.429,E2 -18610.429} C_VEL
LIN {X 0,Y 260.438,Z 577.466,A -85,B 0,C 180,E1 -18612.327,E2 -18612.327} C_VEL
LIN {X 0,Y 258.641,Z 585.136,A -85,B 0,C 180,E1 -18614.637,E2 -18614.637} C_VEL
LIN {X 0,Y 256.917,Z 592.176,A -85,B 0,C 180,E1 -18617.359,E2 -18617.359} C_VEL
LIN {X 0,Y 255.798,Z 596.862,A -85,B 0,C 180,E1 -18619.713,E2 -18619.713} C_VEL
LIN {X 0,Y 255.035,Z 600.444,A -85,B 0,C 180,E1 -18622.081,E2 -18622.081} C_VEL
LIN {X 0,Y 254.694,Z 602.292,A -85,B 0,C 180,E1 -18623.663,E2 -18623.663} C_VEL
LIN {X 0,Y 254.464,Z 603.681,A -85,B 0,C 180,E1 -18625.247,E2 -18625.247} C_VEL
LIN {X 0,Y 254.295,Z 604.669,A -85,B 0,C 180,E1 -18626.831,E2 -18626.831} C_VEL
LIN {X 0,Y 254.113,Z 605.508,A -85,B 0,C 180,E1 -18630,E2 -18630} C_VEL
LIN {X 0,Y 254.145,Z 605.315,A -85,B 0,C 180,E1 -18631.585,E2 -18631.585} C_VEL
LIN {X 0,Y 254.295,Z 604.729,A -85,B 0,C 180,E1 -18633.169,E2 -18633.169} C_VEL
LIN {X 0,Y 254.465,Z 603.764,A -85,B 0,C 180,E1 -18634.753,E2 -18634.753} C_VEL
LIN {X 0,Y 254.829,Z 601.853,A -85,B 0,C 180,E1 -18636.851,E2 -18636.851} C_VEL
LIN {X 0,Y 255.497,Z 598.36,A -85,B 0,C 180,E1 -18639.5,E2 -18639.5} C_VEL
LIN {X 0,Y 256.456,Z 594.116,A -85,B 0,C 180,E1 -18641.86,E2 -18641.86} C_VEL
LIN {X 0,Y 258.037,Z 587.684,A -85,B 0,C 180,E1 -18644.592,E2 -18644.592} C_VEL
LIN {X 0,Y 259.658,Z 580.616,A -85,B 0,C 180,E1 -18646.915,E2 -18646.915} C_VEL
LIN {X 0,Y 261.814,Z 571.799,A -85,B 0,C 180,E1 -18649.197,E2 -18649.197} C_VEL
LIN {X 0,Y 263.617,Z 562.841,A -85,B 0,C 180,E1 -18651.076,E2 -18651.076} C_VEL
LIN {X 0,Y 265.507,Z 552.732,A -85,B 0,C 180,E1 -18652.775,E2 -18652.775} C_VEL
LIN {X 0,Y 267.476,Z 541.573,A -85,B 0,C 180,E1 -18654.239,E2 -18654.239} C_VEL
LIN {X 0,Y 269.277,Z 529.043,A -85,B 0,C 180,E1 -18655.508,E2 -18655.508} C_VEL
LIN {X 0,Y 270.546,Z 516.1,A -85,B 0,C 180,E1 -18656.465,E2 -18656.465} C_VEL
LIN {X 0,Y 271.599,Z 503.308,A -85,B 0,C 180,E1 -18657.081,E2 -18657.081} C_VEL
LIN {X 0,Y 272.326,Z 480.508,A -85,B 0,C 180,E1 -18657.728,E2 -18657.728} C_VEL
LIN {X 0,Y 273.753,Z 434.388,A -85,B 0,C 180,E1 -18658.918,E2 -18658.918} C_VEL
LIN {X 0,Y 267.114,Z 417.699,A -85,B 0,C 180,E1 -18660.224,E2 -18660.224} C_VEL
LIN {X 0,Y 259.96,Z 402.798,A -85,B 0,C 180,E1 -18661.63,E2 -18661.63} C_VEL
LIN {X 0,Y 256.303,Z 395.537,A -85,B 0,C 180,E1 -18662.406,E2 -18662.406} C_VEL
LIN {X 0,Y 256.112,Z 394.58,A -85,B 0,C 180,E1 -18662.967,E2 -18662.967} C_VEL
LIN {X 0,Y 256.128,Z 394.582,A -85,B 0,C 180,E1 -18667.274,E2 -18667.274} C_VEL
LIN {X 0,Y 256.06,Z 394.589,A -85,B 0,C 180,E1 -18671.201,E2 -18671.201} C_VEL
LIN {X 0,Y 256.074,Z 394.581,A -85,B 0,C 180,E1 -18675.525,E2 -18675.525} C_VEL
LIN {X 0,Y 256.101,Z 394.577,A -85,B 0,C 180,E1 -18678.805,E2 -18678.805} C_VEL
LIN {X 0,Y 256.153,Z 394.571,A -85,B 0,C 180,E1 -18682.871,E2 -18682.871} C_VEL
LIN {X 0,Y 256.082,Z 394.58,A -85,B 0,C 180,E1 -18686.709,E2 -18686.709} C_VEL
LIN {X 0,Y 256.134,Z 394.574,A -85,B 0,C 180,E1 -18691.404,E2 -18691.404} C_VEL
LIN {X 0,Y 256.163,Z 394.571,A -85,B 0,C 180,E1 -18695.698,E2 -18695.698} C_VEL
LIN {X 0,Y 256.162,Z 394.576,A -85,B 0,C 180,E1 -18699.104,E2 -18699.104} C_VEL
LIN {X 0,Y 256.29,Z 394.557,A -85,B 0,C 180,E1 -18704.084,E2 -18704.084} C_VEL
LIN {X 0,Y 256.305,Z 394.55,A -85,B 0,C 180,E1 -18708.934,E2 -18708.934} C_VEL
LIN {X 0,Y 256.534,Z 394.529,A -85,B 0,C 180,E1 -18712.127,E2 -18712.127} C_VEL
LIN {X 0,Y 256.709,Z 394.507,A -85,B 0,C 180,E1 -18718.431,E2 -18718.431} C_VEL
LIN {X 0,Y 256.71,Z 394.497,A -85,B 0,C 180,E1 -18721.569,E2 -18721.569} C_VEL
LIN {X 0,Y 256.517,Z 394.523,A -85,B 0,C 180,E1 -18722.881,E2 -18722.881} C_VEL
LIN {X 0,Y 255.794,Z 394.621,A -85,B 0,C 180,E1 -18724.19,E2 -18724.19} C_VEL
LIN {X 0,Y 252.992,Z 394.976,A -85,B 0,C 180,E1 -18726.328,E2 -18726.328} C_VEL
LIN {X 0,Y 249.763,Z 395.372,A -85,B 0,C 180,E1 -18728.958,E2 -18728.958} C_VEL
LIN {X 0,Y 249.365,Z 395.418,A -85,B 0,C 180,E1 -18729.868,E2 -18729.868} C_VEL
LIN {X 0,Y 249.2,Z 395.435,A -85,B 0,C 180,E1 -18734.704,E2 -18734.704} C_VEL
LIN {X 0,Y 249.134,Z 395.45,A -85,B 0,C 180,E1 -18738.078,E2 -18738.078} C_VEL
LIN {X 0,Y 249.083,Z 395.457,A -85,B 0,C 180,E1 -18741.519,E2 -18741.519} C_VEL
LIN {X 0,Y 249.127,Z 395.449,A -85,B 0,C 180,E1 -18745.483,E2 -18745.483} C_VEL
LIN {X 0,Y 249.08,Z 395.458,A -85,B 0,C 180,E1 -18748.994,E2 -18748.994} C_VEL
LIN {X 0,Y 249.032,Z 395.461,A -85,B 0,C 180,E1 -18752.426,E2 -18752.426} C_VEL
LIN {X 0,Y 249.071,Z 395.455,A -85,B 0,C 180,E1 -18756.339,E2 -18756.339} C_VEL
LIN {X 0,Y 249.075,Z 395.453,A -85,B 0,C 180,E1 -18760.465,E2 -18760.465} C_VEL
LIN {X 0,Y 249.018,Z 395.466,A -85,B 0,C 180,E1 -18764.876,E2 -18764.876} C_VEL
LIN {X 0,Y 249.049,Z 395.463,A -85,B 0,C 180,E1 -18767.371,E2 -18767.371} C_VEL
LIN {X 0,Y 249.066,Z 395.546,A -85,B 0,C 180,E1 -18770.458,E2 -18770.458} C_VEL
LIN {X 0,Y 251.236,Z 404.099,A -85,B 0,C 180,E1 -18774.217,E2 -18774.217} C_VEL
LIN {X 0,Y 252.823,Z 411.364,A -85,B 0,C 180,E1 -18777.158,E2 -18777.158} C_VEL
LIN {X 0,Y 260.081,Z 427.82,A -85,B 0,C 180,E1 -18778.696,E2 -18778.696} C_VEL
LIN {X 0,Y 262.373,Z 433.884,A -85,B 0,C 180,E1 -18779.186,E2 -18779.186} C_VEL
LIN {X 0,Y 266.491,Z 461.476,A -85,B 0,C 180,E1 -18780.545,E2 -18780.545} C_VEL
LIN {X 0,Y 266.552,Z 467.538,A -85,B 0,C 180,E1 -18780.736,E2 -18780.736} C_VEL
LIN {X 0,Y 264.773,Z 520.245,A -85,B 0,C 180,E1 -18782.161,E2 -18782.161} C_VEL
LIN {X 0,Y 263.531,Z 534.146,A -85,B 0,C 180,E1 -18782.826,E2 -18782.826} C_VEL
LIN {X 0,Y 261.97,Z 546.589,A -85,B 0,C 180,E1 -18783.727,E2 -18783.727} C_VEL
LIN {X 0,Y 260.191,Z 557.691,A -85,B 0,C 180,E1 -18784.823,E2 -18784.823} C_VEL
LIN {X 0,Y 258.027,Z 569.266,A -85,B 0,C 180,E1 -18786.313,E2 -18786.313} C_VEL
LIN {X 0,Y 255.782,Z 579.692,A -85,B 0,C 180,E1 -18788.015,E2 -18788.015} C_VEL
LIN {X 0,Y 253.855,Z 588.223,A -85,B 0,C 180,E1 -18789.754,E2 -18789.754} C_VEL
LIN {X 0,Y 252.246,Z 596.093,A -85,B 0,C 180,E1 -18791.73,E2 -18791.73} C_VEL
LIN {X 0,Y 250.417,Z 603.803,A -85,B 0,C 180,E1 -18794.12,E2 -18794.12} C_VEL
LIN {X 0,Y 248.654,Z 610.903,A -85,B 0,C 180,E1 -18796.932,E2 -18796.932} C_VEL
LIN {X 0,Y 247.794,Z 615.639,A -85,B 0,C 180,E1 -18799.377,E2 -18799.377} C_VEL
LIN {X 0,Y 247.258,Z 619.261,A -85,B 0,C 180,E1 -18801.83,E2 -18801.83} C_VEL
LIN {X 0,Y 247.008,Z 621.129,A -85,B 0,C 180,E1 -18803.465,E2 -18803.465} C_VEL
LIN {X 0,Y 246.902,Z 622.532,A -85,B 0,C 180,E1 -18805.101,E2 -18805.101} C_VEL
LIN {X 0,Y 246.899,Z 623.537,A -85,B 0,C 180,E1 -18806.736,E2 -18806.736} C_VEL
LIN {X 0,Y 246.982,Z 624.151,A -85,B 0,C 180,E1 -18808.369,E2 -18808.369} C_VEL
LIN {X 0,Y 247.029,Z 624.367,A -85,B 0,C 180,E1 -18810,E2 -18810} C_VEL
LIN {X 0,Y 246.982,Z 624.142,A -85,B 0,C 180,E1 -18811.631,E2 -18811.631} C_VEL
LIN {X 0,Y 246.922,Z 622.512,A -85,B 0,C 180,E1 -18814.898,E2 -18814.898} C_VEL
LIN {X 0,Y 247.005,Z 621.098,A -85,B 0,C 180,E1 -18816.535,E2 -18816.535} C_VEL
LIN {X 0,Y 247.4,Z 618.138,A -85,B 0,C 180,E1 -18818.989,E2 -18818.989} C_VEL
LIN {X 0,Y 248.061,Z 614.137,A -85,B 0,C 180,E1 -18821.439,E2 -18821.439} C_VEL
LIN {X 0,Y 249.36,Z 607.995,A -85,B 0,C 180,E1 -18824.277,E2 -18824.277} C_VEL
LIN {X 0,Y 250.914,Z 601.295,A -85,B 0,C 180,E1 -18826.684,E2 -18826.684} C_VEL
LIN {X 0,Y 252.647,Z 594.092,A -85,B 0,C 180,E1 -18828.767,E2 -18828.767} C_VEL
LIN {X 0,Y 254.693,Z 584.47,A -85,B 0,C 180,E1 -18831.021,E2 -18831.021} C_VEL
LIN {X 0,Y 257.058,Z 573.961,A -85,B 0,C 180,E1 -18832.929,E2 -18832.929} C_VEL
LIN {X 0,Y 259.089,Z 563.562,A -85,B 0,C 180,E1 -18834.435,E2 -18834.435} C_VEL
LIN {X 0,Y 261.026,Z 552.158,A -85,B 0,C 180,E1 -18835.731,E2 -18835.731} C_VEL
LIN {X 0,Y 262.714,Z 540.424,A -85,B 0,C 180,E1 -18836.728,E2 -18836.728} C_VEL
LIN {X 0,Y 264.17,Z 526.894,A -85,B 0,C 180,E1 -18837.531,E2 -18837.531} C_VEL
LIN {X 0,Y 265.021,Z 513.326,A -85,B 0,C 180,E1 -18838.026,E2 -18838.026} C_VEL
LIN {X 0,Y 266.625,Z 463.319,A -85,B 0,C 180,E1 -18839.343,E2 -18839.343} C_VEL
LIN {X 0,Y 262.915,Z 437.208,A -85,B 0,C 180,E1 -18840.599,E2 -18840.599} C_VEL
LIN {X 0,Y 261.818,Z 432.092,A -85,B 0,C 180,E1 -18840.9,E2 -18840.9} C_VEL
LIN {X 0,Y 255.966,Z 418.373,A -85,B 0,C 180,E1 -18842.12,E2 -18842.12} C_VEL
LIN {X 0,Y 252.784,Z 411.167,A -85,B 0,C 180,E1 -18842.824,E2 -18842.824} C_VEL
LIN {X 0,Y 250.764,Z 402.184,A -85,B 0,C 180,E1 -18846.552,E2 -18846.552} C_VEL
LIN {X 0,Y 249.067,Z 395.461,A -85,B 0,C 180,E1 -18849.542,E2 -18849.542} C_VEL
LIN {X 0,Y 249.043,Z 395.462,A -85,B 0,C 180,E1 -18852.801,E2 -18852.801} C_VEL
LIN {X 0,Y 249.06,Z 395.457,A -85,B 0,C 180,E1 -18857.372,E2 -18857.372} C_VEL
LIN {X 0,Y 249.049,Z 395.462,A -85,B 0,C 180,E1 -18861.624,E2 -18861.624} C_VEL
LIN {X 0,Y 249.058,Z 395.458,A -85,B 0,C 180,E1 -18865.642,E2 -18865.642} C_VEL
LIN {X 0,Y 249.048,Z 395.461,A -85,B 0,C 180,E1 -18869.473,E2 -18869.473} C_VEL
LIN {X 0,Y 249.07,Z 395.456,A -85,B 0,C 180,E1 -18873.162,E2 -18873.162} C_VEL
LIN {X 0,Y 249.074,Z 395.448,A -85,B 0,C 180,E1 -18876.732,E2 -18876.732} C_VEL
LIN {X 0,Y 249.106,Z 395.453,A -85,B 0,C 180,E1 -18880.211,E2 -18880.211} C_VEL
LIN {X 0,Y 249.238,Z 395.43,A -85,B 0,C 180,E1 -18883.622,E2 -18883.622} C_VEL
LIN {X 0,Y 249.248,Z 395.431,A -85,B 0,C 180,E1 -18888.616,E2 -18888.616} C_VEL
LIN {X 0,Y 249.476,Z 395.406,A -85,B 0,C 180,E1 -18891.903,E2 -18891.903} C_VEL
LIN {X 0,Y 249.431,Z 395.402,A -85,B 0,C 180,E1 -18896.77,E2 -18896.77} C_VEL
LIN {X 0,Y 249.73,Z 395.375,A -85,B 0,C 180,E1 -18900,E2 -18900} C_VEL
LIN {X 0,Y 249.431,Z 395.406,A -85,B 0,C 180,E1 -18903.231,E2 -18903.231} C_VEL
